LIN {X 0,Y 306.825,Z 754.98,A -85,B 0,C 180,E1 -15915.408,E2 -15915.408} C_VEL
LIN {X 0,Y 305.546,Z 762.411,A -85,B 0,C 180,E1 -15917.38,E2 -15917.38} C_VEL
LIN {X 0,Y 304.708,Z 768.383,A -85,B 0,C 180,E1 -15919.368,E2 -15919.368} C_VEL
LIN {X 0,Y 304.145,Z 773.106,A -85,B 0,C 180,E1 -15921.363,E2 -15921.363} C_VEL
LIN {X 0,Y 303.739,Z 776.717,A -85,B 0,C 180,E1 -15923.358,E2 -15923.358} C_VEL
LIN {X 0,Y 303.637,Z 778.581,A -85,B 0,C 180,E1 -15924.689,E2 -15924.689} C_VEL
LIN {X 0,Y 303.631,Z 779.979,A -85,B 0,C 180,E1 -15926.019,E2 -15926.019} C_VEL
LIN {X 0,Y 303.607,Z 780.975,A -85,B 0,C 180,E1 -15927.348,E2 -15927.348} C_VEL
LIN {X 0,Y 303.564,Z 781.589,A -85,B 0,C 180,E1 -15928.675,E2 -15928.675} C_VEL
LIN {X 0,Y 303.543,Z 783.849,A -85,B 0,C 180,E1 -15931.328,E2 -15931.328} C_VEL
LIN {X 0,Y 303.613,Z 784.204,A -85,B 0,C 180,E1 -15932.655,E2 -15932.655} C_VEL
LIN {X 0,Y 303.689,Z 783.949,A -85,B 0,C 180,E1 -15933.982,E2 -15933.982} C_VEL
LIN {X 0,Y 303.902,Z 782.447,A -85,B 0,C 180,E1 -15936.058,E2 -15936.058} C_VEL
LIN {X 0,Y 304.24,Z 779.671,A -85,B 0,C 180,E1 -15937.968,E2 -15937.968} C_VEL
LIN {X 0,Y 304.907,Z 775.432,A -85,B 0,C 180,E1 -15939.956,E2 -15939.956} C_VEL
LIN {X 0,Y 305.723,Z 769.513,A -85,B 0,C 180,E1 -15941.941,E2 -15941.941} C_VEL
LIN {X 0,Y 306.312,Z 764.494,A -85,B 0,C 180,E1 -15943.265,E2 -15943.265} C_VEL
LIN {X 0,Y 307.414,Z 756.689,A -85,B 0,C 180,E1 -15944.905,E2 -15944.905} C_VEL
LIN {X 0,Y 308.373,Z 747.222,A -85,B 0,C 180,E1 -15946.483,E2 -15946.483} C_VEL
LIN {X 0,Y 308.794,Z 741.989,A -85,B 0,C 180,E1 -15947.211,E2 -15947.211} C_VEL
LIN {X 0,Y 310.204,Z 732.695,A -85,B 0,C 180,E1 -15948.665,E2 -15948.665} C_VEL
LIN {X 0,Y 311.896,Z 721.129,A -85,B 0,C 180,E1 -15950.099,E2 -15950.099} C_VEL
LIN {X 0,Y 313.363,Z 709.743,A -85,B 0,C 180,E1 -15951.202,E2 -15951.202} C_VEL
LIN {X 0,Y 314.572,Z 698.034,A -85,B 0,C 180,E1 -15952.063,E2 -15952.063} C_VEL
LIN {X 0,Y 315.64,Z 685.44,A -85,B 0,C 180,E1 -15952.718,E2 -15952.718} C_VEL
LIN {X 0,Y 316.262,Z 672.598,A -85,B 0,C 180,E1 -15953.146,E2 -15953.146} C_VEL
LIN {X 0,Y 317.533,Z 619.147,A -85,B 0,C 180,E1 -15954.372,E2 -15954.372} C_VEL
LIN {X 0,Y 319.338,Z 611.037,A -85,B 0,C 180,E1 -15955.032,E2 -15955.032} C_VEL
LIN {X 0,Y 321.692,Z 593.032,A -85,B 0,C 180,E1 -15957.134,E2 -15957.134} C_VEL
LIN {X 0,Y 321.832,Z 587.078,A -85,B 0,C 180,E1 -15958.099,E2 -15958.099} C_VEL
LIN {X 0,Y 321.31,Z 583.094,A -85,B 0,C 180,E1 -15958.964,E2 -15958.964} C_VEL
LIN {X 0,Y 320.097,Z 575.053,A -85,B 0,C 180,E1 -15961.099,E2 -15961.099} C_VEL
LIN {X 0,Y 319.576,Z 571.128,A -85,B 0,C 180,E1 -15962.355,E2 -15962.355} C_VEL
LIN {X 0,Y 318.499,Z 569.11,A -85,B 0,C 180,E1 -15963.481,E2 -15963.481} C_VEL
LIN {X 0,Y 317.152,Z 566.664,A -85,B 0,C 180,E1 -15965.181,E2 -15965.181} C_VEL
LIN {X 0,Y 316.078,Z 565.019,A -85,B 0,C 180,E1 -15966.896,E2 -15966.896} C_VEL
LIN {X 0,Y 315.22,Z 564.079,A -85,B 0,C 180,E1 -15968.708,E2 -15968.708} C_VEL
LIN {X 0,Y 314.759,Z 563.673,A -85,B 0,C 180,E1 -15970.61,E2 -15970.61} C_VEL
LIN {X 0,Y 314.997,Z 564.269,A -85,B 0,C 180,E1 -15973.762,E2 -15973.762} C_VEL
LIN {X 0,Y 315.704,Z 566.324,A -85,B 0,C 180,E1 -15976.362,E2 -15976.362} C_VEL
LIN {X 0,Y 316.93,Z 569.514,A -85,B 0,C 180,E1 -15978.936,E2 -15978.936} C_VEL
LIN {X 0,Y 318.658,Z 574.729,A -85,B 0,C 180,E1 -15981.863,E2 -15981.863} C_VEL
LIN {X 0,Y 320.123,Z 580.476,A -85,B 0,C 180,E1 -15984.323,E2 -15984.323} C_VEL
LIN {X 0,Y 321.256,Z 585.775,A -85,B 0,C 180,E1 -15986.235,E2 -15986.235} C_VEL
LIN {X 0,Y 322.064,Z 591.78,A -85,B 0,C 180,E1 -15988.104,E2 -15988.104} C_VEL
LIN {X 0,Y 321.886,Z 594.252,A -85,B 0,C 180,E1 -15988.719,E2 -15988.719} C_VEL
LIN {X 0,Y 317.742,Z 616.41,A -85,B 0,C 180,E1 -15993.422,E2 -15993.422} C_VEL
LIN {X 0,Y 315.354,Z 632.652,A -85,B 0,C 180,E1 -15996.739,E2 -15996.739} C_VEL
LIN {X 0,Y 318.091,Z 647.204,A -85,B 0,C 180,E1 -15997.92,E2 -15997.92} C_VEL
LIN {X 0,Y 319.528,Z 659.288,A -85,B 0,C 180,E1 -15998.728,E2 -15998.728} C_VEL
LIN {X 0,Y 316.266,Z 706.91,A -85,B 0,C 180,E1 -16000.529,E2 -16000.529} C_VEL
LIN {X 0,Y 315.093,Z 718.743,A -85,B 0,C 180,E1 -16001.215,E2 -16001.215} C_VEL
LIN {X 0,Y 313.817,Z 728.863,A -85,B 0,C 180,E1 -16002.065,E2 -16002.065} C_VEL
LIN {X 0,Y 312.287,Z 738.973,A -85,B 0,C 180,E1 -16003.157,E2 -16003.157} C_VEL
LIN {X 0,Y 310.981,Z 746.942,A -85,B 0,C 180,E1 -16004.265,E2 -16004.265} C_VEL
LIN {X 0,Y 309.584,Z 754.286,A -85,B 0,C 180,E1 -16005.539,E2 -16005.539} C_VEL
LIN {X 0,Y 308.32,Z 760.339,A -85,B 0,C 180,E1 -16006.824,E2 -16006.824} C_VEL
LIN {X 0,Y 307.008,Z 766.483,A -85,B 0,C 180,E1 -16008.445,E2 -16008.445} C_VEL
LIN {X 0,Y 305.966,Z 771.229,A -85,B 0,C 180,E1 -16010.08,E2 -16010.08} C_VEL
LIN {X 0,Y 305.24,Z 774.224,A -85,B 0,C 180,E1 -16011.393,E2 -16011.393} C_VEL
LIN {X 0,Y 304.609,Z 777.366,A -85,B 0,C 180,E1 -16013.376,E2 -16013.376} C_VEL
LIN {X 0,Y 304.172,Z 778.748,A -85,B 0,C 180,E1 -16014.697,E2 -16014.697} C_VEL
LIN {X 0,Y 303.852,Z 779.547,A -85,B 0,C 180,E1 -16016.021,E2 -16016.021} C_VEL
LIN {X 0,Y 303.664,Z 779.771,A -85,B 0,C 180,E1 -16017.347,E2 -16017.347} C_VEL
LIN {X 0,Y 303.55,Z 779.388,A -85,B 0,C 180,E1 -16018.673,E2 -16018.673} C_VEL
LIN {X 0,Y 303.534,Z 778.387,A -85,B 0,C 180,E1 -16020,E2 -16020} C_VEL
LIN {X 0,Y 303.571,Z 775.717,A -85,B 0,C 180,E1 -16021.99,E2 -16021.99} C_VEL
LIN {X 0,Y 303.815,Z 771.583,A -85,B 0,C 180,E1 -16023.979,E2 -16023.979} C_VEL
LIN {X 0,Y 303.878,Z 765.594,A -85,B 0,C 180,E1 -16026.01,E2 -16026.01} C_VEL
LIN {X 0,Y 304.246,Z 759.517,A -85,B 0,C 180,E1 -16027.571,E2 -16027.571} C_VEL
LIN {X 0,Y 304.58,Z 752.814,A -85,B 0,C 180,E1 -16028.961,E2 -16028.961} C_VEL
LIN {X 0,Y 305.028,Z 744.827,A -85,B 0,C 180,E1 -16030.286,E2 -16030.286} C_VEL
LIN {X 0,Y 305.485,Z 736.01,A -85,B 0,C 180,E1 -16031.445,E2 -16031.445} C_VEL
LIN {X 0,Y 305.984,Z 726.568,A -85,B 0,C 180,E1 -16032.435,E2 -16032.435} C_VEL
LIN {X 0,Y 306.384,Z 715.842,A -85,B 0,C 180,E1 -16033.261,E2 -16033.261} C_VEL
LIN {X 0,Y 306.839,Z 705.379,A -85,B 0,C 180,E1 -16033.832,E2 -16033.832} C_VEL
LIN {X 0,Y 307.924,Z 653.383,A -85,B 0,C 180,E1 -16035.606,E2 -16035.606} C_VEL
LIN {X 0,Y 306.354,Z 631.88,A -85,B 0,C 180,E1 -16036.403,E2 -16036.403} C_VEL
LIN {X 0,Y 307.681,Z 611.142,A -85,B 0,C 180,E1 -16040.383,E2 -16040.383} C_VEL
LIN {X 0,Y 309.256,Z 588.247,A -85,B 0,C 180,E1 -16044.799,E2 -16044.799} C_VEL
LIN {X 0,Y 310.552,Z 571.445,A -85,B 0,C 180,E1 -16048.041,E2 -16048.041} C_VEL
LIN {X 0,Y 308.725,Z 561.43,A -85,B 0,C 180,E1 -16050.11,E2 -16050.11} C_VEL
LIN {X 0,Y 305.543,Z 546.572,A -85,B 0,C 180,E1 -16053.314,E2 -16053.314} C_VEL
LIN {X 0,Y 305.48,Z 546.435,A -85,B 0,C 180,E1 -16056.739,E2 -16056.739} C_VEL
LIN {X 0,Y 305.459,Z 546.414,A -85,B 0,C 180,E1 -16060.599,E2 -16060.599} C_VEL
LIN {X 0,Y 305.431,Z 546.409,A -85,B 0,C 180,E1 -16064.494,E2 -16064.494} C_VEL
LIN {X 0,Y 305.48,Z 546.425,A -85,B 0,C 180,E1 -16068.149,E2 -16068.149} C_VEL
LIN {X 0,Y 305.472,Z 546.41,A -85,B 0,C 180,E1 -16071.596,E2 -16071.596} C_VEL
LIN {X 0,Y 305.467,Z 546.424,A -85,B 0,C 180,E1 -16074.886,E2 -16074.886} C_VEL
LIN {X 0,Y 305.456,Z 546.43,A -85,B 0,C 180,E1 -16078.354,E2 -16078.354} C_VEL
LIN {X 0,Y 305.535,Z 546.476,A -85,B 0,C 180,E1 -16080.803,E2 -16080.803} C_VEL
LIN {X 0,Y 307.121,Z 553.574,A -85,B 0,C 180,E1 -16083.444,E2 -16083.444} C_VEL
LIN {X 0,Y 307.557,Z 555.026,A -85,B 0,C 180,E1 -16083.632,E2 -16083.632} C_VEL
LIN {X 0,Y 314.364,Z 571.514,A -85,B 0,C 180,E1 -16084.671,E2 -16084.671} C_VEL
LIN {X 0,Y 316.455,Z 577.195,A -85,B 0,C 180,E1 -16084.992,E2 -16084.992} C_VEL
LIN {X 0,Y 318.23,Z 587.121,A -85,B 0,C 180,E1 -16085.384,E2 -16085.384} C_VEL
LIN {X 0,Y 316.373,Z 660.195,A -85,B 0,C 180,E1 -16087.036,E2 -16087.036} C_VEL
LIN {X 0,Y 315.644,Z 673.592,A -85,B 0,C 180,E1 -16087.585,E2 -16087.585} C_VEL
LIN {X 0,Y 314.69,Z 686.351,A -85,B 0,C 180,E1 -16088.376,E2 -16088.376} C_VEL
LIN {X 0,Y 313.452,Z 697.672,A -85,B 0,C 180,E1 -16089.32,E2 -16089.32} C_VEL
LIN {X 0,Y 311.954,Z 709.318,A -85,B 0,C 180,E1 -16090.59,E2 -16090.59} C_VEL
LIN {X 0,Y 310.534,Z 720.204,A -85,B 0,C 180,E1 -16092.108,E2 -16092.108} C_VEL
LIN {X 0,Y 309.013,Z 729.997,A -85,B 0,C 180,E1 -16093.822,E2 -16093.822} C_VEL
LIN {X 0,Y 307.427,Z 738.909,A -85,B 0,C 180,E1 -16095.773,E2 -16095.773} C_VEL
LIN {X 0,Y 306.273,Z 746.076,A -85,B 0,C 180,E1 -16097.744,E2 -16097.744} C_VEL
LIN {X 0,Y 305.411,Z 750.913,A -85,B 0,C 180,E1 -16099.391,E2 -16099.391} C_VEL
LIN {X 0,Y 304.679,Z 755.609,A -85,B 0,C 180,E1 -16101.376,E2 -16101.376} C_VEL
LIN {X 0,Y 304.196,Z 759.318,A -85,B 0,C 180,E1 -16103.442,E2 -16103.442} C_VEL
LIN {X 0,Y 304.024,Z 761.05,A -85,B 0,C 180,E1 -16104.693,E2 -16104.693} C_VEL
LIN {X 0,Y 303.867,Z 762.446,A -85,B 0,C 180,E1 -16106.02,E2 -16106.02} C_VEL
LIN {X 0,Y 303.617,Z 764.054,A -85,B 0,C 180,E1 -16108.672,E2 -16108.672} C_VEL
LIN {X 0,Y 303.611,Z 764.285,A -85,B 0,C 180,E1 -16109.999,E2 -16109.999} C_VEL
LIN {X 0,Y 303.617,Z 764.095,A -85,B 0,C 180,E1 -16111.325,E2 -16111.325} C_VEL
LIN {X 0,Y 303.862,Z 762.543,A -85,B 0,C 180,E1 -16113.978,E2 -16113.978} C_VEL
LIN {X 0,Y 304.019,Z 761.188,A -85,B 0,C 180,E1 -16115.304,E2 -16115.304} C_VEL
LIN {X 0,Y 304.345,Z 758.321,A -85,B 0,C 180,E1 -16117.295,E2 -16117.295} C_VEL
LIN {X 0,Y 304.844,Z 754.433,A -85,B 0,C 180,E1 -16119.286,E2 -16119.286} C_VEL
LIN {X 0,Y 305.715,Z 749.416,A -85,B 0,C 180,E1 -16121.267,E2 -16121.267} C_VEL
LIN {X 0,Y 306.746,Z 743.101,A -85,B 0,C 180,E1 -16123.244,E2 -16123.244} C_VEL
LIN {X 0,Y 308.104,Z 735.191,A -85,B 0,C 180,E1 -16125.206,E2 -16125.206} C_VEL
LIN {X 0,Y 309.826,Z 725.349,A -85,B 0,C 180,E1 -16127.149,E2 -16127.149} C_VEL
LIN {X 0,Y 311.239,Z 715.021,A -85,B 0,C 180,E1 -16128.769,E2 -16128.769} C_VEL
LIN {X 0,Y 312.599,Z 704.79,A -85,B 0,C 180,E1 -16130.05,E2 -16130.05} C_VEL
LIN {X 0,Y 313.983,Z 693.583,A -85,B 0,C 180,E1 -16131.156,E2 -16131.156} C_VEL
LIN {X 0,Y 315.21,Z 680.94,A -85,B 0,C 180,E1 -16132.1,E2 -16132.1} C_VEL
LIN {X 0,Y 316.045,Z 668.274,A -85,B 0,C 180,E1 -16132.771,E2 -16132.771} C_VEL
LIN {X 0,Y 316.658,Z 655.229,A -85,B 0,C 180,E1 -16133.199,E2 -16133.199} C_VEL
LIN {X 0,Y 318.19,Z 585.949,A -85,B 0,C 180,E1 -16134.76,E2 -16134.76} C_VEL
LIN {X 0,Y 315.996,Z 575.742,A -85,B 0,C 180,E1 -16135.197,E2 -16135.197} C_VEL
LIN {X 0,Y 309.077,Z 558.611,A -85,B 0,C 180,E1 -16136.241,E2 -16136.241} C_VEL
LIN {X 0,Y 307.194,Z 553.882,A -85,B 0,C 180,E1 -16136.597,E2 -16136.597} C_VEL
LIN {X 0,Y 305.932,Z 548.426,A -85,B 0,C 180,E1 -16138.518,E2 -16138.518} C_VEL
LIN {X 0,Y 305.264,Z 547.176,A -85,B 0,C 180,E1 -16139.189,E2 -16139.189} C_VEL
LIN {X 0,Y 304.227,Z 546.692,A -85,B 0,C 180,E1 -16139.887,E2 -16139.887} C_VEL
LIN {X 0,Y 299.362,Z 547.224,A -85,B 0,C 180,E1 -16142.794,E2 -16142.794} C_VEL
LIN {X 0,Y 298.448,Z 547.31,A -85,B 0,C 180,E1 -16143.945,E2 -16143.945} C_VEL
LIN {X 0,Y 298.4,Z 547.316,A -85,B 0,C 180,E1 -16144.333,E2 -16144.333} C_VEL
LIN {X 0,Y 298.433,Z 547.313,A -85,B 0,C 180,E1 -16147.753,E2 -16147.753} C_VEL
LIN {X 0,Y 298.382,Z 547.313,A -85,B 0,C 180,E1 -16151.26,E2 -16151.26} C_VEL
LIN {X 0,Y 298.35,Z 547.302,A -85,B 0,C 180,E1 -16155.034,E2 -16155.034} C_VEL
LIN {X 0,Y 298.427,Z 547.307,A -85,B 0,C 180,E1 -16156.925,E2 -16156.925} C_VEL
LIN {X 0,Y 298.421,Z 547.286,A -85,B 0,C 180,E1 -16161,E2 -16161} C_VEL
LIN {X 0,Y 298.43,Z 547.307,A -85,B 0,C 180,E1 -16163.932,E2 -16163.932} C_VEL
LIN {X 0,Y 298.39,Z 547.31,A -85,B 0,C 180,E1 -16167.982,E2 -16167.982} C_VEL
LIN {X 0,Y 298.457,Z 547.297,A -85,B 0,C 180,E1 -16171.904,E2 -16171.904} C_VEL
LIN {X 0,Y 298.479,Z 547.304,A -85,B 0,C 180,E1 -16174.923,E2 -16174.923} C_VEL
LIN {X 0,Y 298.443,Z 547.303,A -85,B 0,C 180,E1 -16179.315,E2 -16179.315} C_VEL
LIN {X 0,Y 298.531,Z 547.292,A -85,B 0,C 180,E1 -16182.179,E2 -16182.179} C_VEL
LIN {X 0,Y 298.586,Z 547.281,A -85,B 0,C 180,E1 -16184.994,E2 -16184.994} C_VEL
LIN {X 0,Y 298.586,Z 547.281,A -85,B 0,C 180,E1 -16189.146,E2 -16189.146} C_VEL
LIN {X 0,Y 298.751,Z 547.266,A -85,B 0,C 180,E1 -16191.886,E2 -16191.886} C_VEL
LIN {X 0,Y 298.654,Z 547.28,A -85,B 0,C 180,E1 -16194.599,E2 -16194.599} C_VEL
LIN {X 0,Y 298.918,Z 547.244,A -85,B 0,C 180,E1 -16198.653,E2 -16198.653} C_VEL
LIN {X 0,Y 298.918,Z 547.249,A -85,B 0,C 180,E1 -16201.347,E2 -16201.347} C_VEL
LIN {X 0,Y 298.792,Z 547.264,A -85,B 0,C 180,E1 -16206.754,E2 -16206.754} C_VEL
LIN {X 0,Y 298.673,Z 547.268,A -85,B 0,C 180,E1 -16209.481,E2 -16209.481} C_VEL
LIN {X 0,Y 298.546,Z 547.297,A -85,B 0,C 180,E1 -16213.616,E2 -16213.616} C_VEL
LIN {X 0,Y 298.541,Z 547.285,A -85,B 0,C 180,E1 -16216.409,E2 -16216.409} C_VEL
LIN {X 0,Y 298.509,Z 547.301,A -85,B 0,C 180,E1 -16219.658,E2 -16219.658} C_VEL
LIN {X 0,Y 298.451,Z 547.308,A -85,B 0,C 180,E1 -16223.598,E2 -16223.598} C_VEL
LIN {X 0,Y 298.477,Z 547.295,A -85,B 0,C 180,E1 -16226.576,E2 -16226.576} C_VEL
LIN {X 0,Y 298.41,Z 547.313,A -85,B 0,C 180,E1 -16229.642,E2 -16229.642} C_VEL
LIN {X 0,Y 298.389,Z 547.315,A -85,B 0,C 180,E1 -16232.801,E2 -16232.801} C_VEL
LIN {X 0,Y 298.441,Z 547.284,A -85,B 0,C 180,E1 -16236.809,E2 -16236.809} C_VEL
LIN {X 0,Y 298.409,Z 547.305,A -85,B 0,C 180,E1 -16241.258,E2 -16241.258} C_VEL
LIN {X 0,Y 298.412,Z 547.314,A -85,B 0,C 180,E1 -16245.048,E2 -16245.048} C_VEL
LIN {X 0,Y 298.45,Z 547.309,A -85,B 0,C 180,E1 -16248.751,E2 -16248.751} C_VEL
LIN {X 0,Y 298.463,Z 547.279,A -85,B 0,C 180,E1 -16253.189,E2 -16253.189} C_VEL
LIN {X 0,Y 298.426,Z 547.398,A -85,B 0,C 180,E1 -16255.789,E2 -16255.789} C_VEL
LIN {X 0,Y 300.553,Z 556.606,A -85,B 0,C 180,E1 -16259.042,E2 -16259.042} C_VEL
LIN {X 0,Y 302.687,Z 566.604,A -85,B 0,C 180,E1 -16262.332,E2 -16262.332} C_VEL
LIN {X 0,Y 303.149,Z 569.151,A -85,B 0,C 180,E1 -16263.067,E2 -16263.067} C_VEL
LIN {X 0,Y 305.199,Z 575.225,A -85,B 0,C 180,E1 -16263.464,E2 -16263.464} C_VEL
LIN {X 0,Y 310.189,Z 604.18,A -85,B 0,C 180,E1 -16264.648,E2 -16264.648} C_VEL
LIN {X 0,Y 311.262,Z 612.409,A -85,B 0,C 180,E1 -16264.946,E2 -16264.946} C_VEL
LIN {X 0,Y 309.607,Z 677.501,A -85,B 0,C 180,E1 -16266.462,E2 -16266.462} C_VEL
LIN {X 0,Y 308.607,Z 691.422,A -85,B 0,C 180,E1 -16267.047,E2 -16267.047} C_VEL
LIN {X 0,Y 307.431,Z 703.883,A -85,B 0,C 180,E1 -16267.841,E2 -16267.841} C_VEL
LIN {X 0,Y 306.08,Z 715.003,A -85,B 0,C 180,E1 -16268.8,E2 -16268.8} C_VEL
LIN {X 0,Y 304.44,Z 726.577,A -85,B 0,C 180,E1 -16270.094,E2 -16270.094} C_VEL
LIN {X 0,Y 302.776,Z 737,A -85,B 0,C 180,E1 -16271.564,E2 -16271.564} C_VEL
LIN {X 0,Y 301.509,Z 745.549,A -85,B 0,C 180,E1 -16273.065,E2 -16273.065} C_VEL
LIN {X 0,Y 300.188,Z 753.4,A -85,B 0,C 180,E1 -16274.73,E2 -16274.73} C_VEL
LIN {X 0,Y 298.808,Z 761.087,A -85,B 0,C 180,E1 -16276.744,E2 -16276.744} C_VEL
LIN {X 0,Y 297.712,Z 768.179,A -85,B 0,C 180,E1 -16279.115,E2 -16279.115} C_VEL
LIN {X 0,Y 297.087,Z 772.901,A -85,B 0,C 180,E1 -16281.156,E2 -16281.156} C_VEL
LIN {X 0,Y 296.686,Z 776.513,A -85,B 0,C 180,E1 -16283.199,E2 -16283.199} C_VEL
LIN {X 0,Y 296.552,Z 778.377,A -85,B 0,C 180,E1 -16284.562,E2 -16284.562} C_VEL
LIN {X 0,Y 296.528,Z 779.774,A -85,B 0,C 180,E1 -16285.924,E2 -16285.924} C_VEL
LIN {X 0,Y 296.533,Z 780.771,A -85,B 0,C 180,E1 -16287.284,E2 -16287.284} C_VEL
LIN {X 0,Y 296.484,Z 781.379,A -85,B 0,C 180,E1 -16288.643,E2 -16288.643} C_VEL
LIN {X 0,Y 296.465,Z 783.587,A -85,B 0,C 180,E1 -16291.36,E2 -16291.36} C_VEL
LIN {X 0,Y 296.541,Z 784.068,A -85,B 0,C 180,E1 -16292.718,E2 -16292.718} C_VEL
LIN {X 0,Y 296.591,Z 783.961,A -85,B 0,C 180,E1 -16294.078,E2 -16294.078} C_VEL
LIN {X 0,Y 296.821,Z 782.819,A -85,B 0,C 180,E1 -16296.033,E2 -16296.033} C_VEL
LIN {X 0,Y 297.23,Z 780.165,A -85,B 0,C 180,E1 -16298.157,E2 -16298.157} C_VEL
LIN {X 0,Y 297.681,Z 777.674,A -85,B 0,C 180,E1 -16299.514,E2 -16299.514} C_VEL
LIN {X 0,Y 298.212,Z 774.484,A -85,B 0,C 180,E1 -16300.869,E2 -16300.869} C_VEL
LIN {X 0,Y 299.015,Z 769.366,A -85,B 0,C 180,E1 -16302.558,E2 -16302.558} C_VEL
LIN {X 0,Y 299.803,Z 764.371,A -85,B 0,C 180,E1 -16303.904,E2 -16303.904} C_VEL
LIN {X 0,Y 300.94,Z 756.662,A -85,B 0,C 180,E1 -16305.58,E2 -16305.58} C_VEL
LIN {X 0,Y 302.009,Z 747.777,A -85,B 0,C 180,E1 -16307.097,E2 -16307.097} C_VEL
LIN {X 0,Y 302.796,Z 738.445,A -85,B 0,C 180,E1 -16308.384,E2 -16308.384} C_VEL
LIN {X 0,Y 303.445,Z 732.497,A -85,B 0,C 180,E1 -16309.097,E2 -16309.097} C_VEL
LIN {X 0,Y 305.028,Z 722.348,A -85,B 0,C 180,E1 -16310.396,E2 -16310.396} C_VEL
LIN {X 0,Y 306.516,Z 711.301,A -85,B 0,C 180,E1 -16311.523,E2 -16311.523} C_VEL
LIN {X 0,Y 307.889,Z 699.055,A -85,B 0,C 180,E1 -16312.48,E2 -16312.48} C_VEL
LIN {X 0,Y 308.997,Z 687.058,A -85,B 0,C 180,E1 -16313.146,E2 -16313.146} C_VEL
LIN {X 0,Y 309.703,Z 673.882,A -85,B 0,C 180,E1 -16313.621,E2 -16313.621} C_VEL
LIN {X 0,Y 310.962,Z 625.82,A -85,B 0,C 180,E1 -16314.761,E2 -16314.761} C_VEL
LIN {X 0,Y 314.172,Z 612.643,A -85,B 0,C 180,E1 -16315.862,E2 -16315.862} C_VEL
LIN {X 0,Y 316.645,Z 596.601,A -85,B 0,C 180,E1 -16317.782,E2 -16317.782} C_VEL
LIN {X 0,Y 316.946,Z 590.536,A -85,B 0,C 180,E1 -16318.788,E2 -16318.788} C_VEL
LIN {X 0,Y 316.071,Z 583.822,A -85,B 0,C 180,E1 -16320.453,E2 -16320.453} C_VEL
LIN {X 0,Y 315.334,Z 577.432,A -85,B 0,C 180,E1 -16322.338,E2 -16322.338} C_VEL
LIN {X 0,Y 315.02,Z 576.052,A -85,B 0,C 180,E1 -16322.881,E2 -16322.881} C_VEL
LIN {X 0,Y 313.397,Z 573.124,A -85,B 0,C 180,E1 -16324.757,E2 -16324.757} C_VEL
LIN {X 0,Y 312.55,Z 571.715,A -85,B 0,C 180,E1 -16325.953,E2 -16325.953} C_VEL
LIN {X 0,Y 311.446,Z 570.264,A -85,B 0,C 180,E1 -16327.833,E2 -16327.833} C_VEL
LIN {X 0,Y 310.711,Z 569.522,A -85,B 0,C 180,E1 -16329.731,E2 -16329.731} C_VEL
LIN {X 0,Y 310.497,Z 569.555,A -85,B 0,C 180,E1 -16332.77,E2 -16332.77} C_VEL
LIN {X 0,Y 310.771,Z 570.278,A -85,B 0,C 180,E1 -16334.513,E2 -16334.513} C_VEL
LIN {X 0,Y 311.578,Z 572.968,A -85,B 0,C 180,E1 -16337.415,E2 -16337.415} C_VEL
LIN {X 0,Y 312.662,Z 576.349,A -85,B 0,C 180,E1 -16339.842,E2 -16339.842} C_VEL
LIN {X 0,Y 313.856,Z 580.516,A -85,B 0,C 180,E1 -16342.117,E2 -16342.117} C_VEL
LIN {X 0,Y 315.36,Z 587.458,A -85,B 0,C 180,E1 -16345.029,E2 -16345.029} C_VEL
LIN {X 0,Y 316.237,Z 593.305,A -85,B 0,C 180,E1 -16347.045,E2 -16347.045} C_VEL
LIN {X 0,Y 316.318,Z 596.748,A -85,B 0,C 180,E1 -16348.053,E2 -16348.053} C_VEL
LIN {X 0,Y 312.172,Z 617.259,A -85,B 0,C 180,E1 -16352.515,E2 -16352.515} C_VEL
LIN {X 0,Y 309.562,Z 632.55,A -85,B 0,C 180,E1 -16355.74,E2 -16355.74} C_VEL
LIN {X 0,Y 312.365,Z 647.726,A -85,B 0,C 180,E1 -16357.07,E2 -16357.07} C_VEL
LIN {X 0,Y 313.908,Z 660.09,A -85,B 0,C 180,E1 -16357.941,E2 -16357.941} C_VEL
LIN {X 0,Y 310.383,Z 707.099,A -85,B 0,C 180,E1 -16359.8,E2 -16359.8} C_VEL
LIN {X 0,Y 309.16,Z 718.874,A -85,B 0,C 180,E1 -16360.495,E2 -16360.495} C_VEL
LIN {X 0,Y 307.79,Z 728.991,A -85,B 0,C 180,E1 -16361.357,E2 -16361.357} C_VEL
LIN {X 0,Y 306.381,Z 737.697,A -85,B 0,C 180,E1 -16362.306,E2 -16362.306} C_VEL
LIN {X 0,Y 304.711,Z 746.945,A -85,B 0,C 180,E1 -16363.588,E2 -16363.588} C_VEL
LIN {X 0,Y 303.217,Z 754.234,A -85,B 0,C 180,E1 -16364.885,E2 -16364.885} C_VEL
LIN {X 0,Y 301.835,Z 760.322,A -85,B 0,C 180,E1 -16366.192,E2 -16366.192} C_VEL
LIN {X 0,Y 300.363,Z 766.508,A -85,B 0,C 180,E1 -16367.843,E2 -16367.843} C_VEL
LIN {X 0,Y 299.433,Z 770.408,A -85,B 0,C 180,E1 -16369.177,E2 -16369.177} C_VEL
LIN {X 0,Y 298.252,Z 774.825,A -85,B 0,C 180,E1 -16371.19,E2 -16371.19} C_VEL
LIN {X 0,Y 297.841,Z 776.718,A -85,B 0,C 180,E1 -16372.335,E2 -16372.335} C_VEL
LIN {X 0,Y 297.119,Z 779.033,A -85,B 0,C 180,E1 -16374.571,E2 -16374.571} C_VEL
LIN {X 0,Y 296.779,Z 779.685,A -85,B 0,C 180,E1 -16375.926,E2 -16375.926} C_VEL
LIN {X 0,Y 296.596,Z 779.76,A -85,B 0,C 180,E1 -16377.284,E2 -16377.284} C_VEL
LIN {X 0,Y 296.473,Z 779.257,A -85,B 0,C 180,E1 -16378.642,E2 -16378.642} C_VEL
LIN {X 0,Y 296.453,Z 778.164,A -85,B 0,C 180,E1 -16380,E2 -16380} C_VEL
LIN {X 0,Y 296.498,Z 775.28,A -85,B 0,C 180,E1 -16382.038,E2 -16382.038} C_VEL
LIN {X 0,Y 296.662,Z 772.566,A -85,B 0,C 180,E1 -16383.395,E2 -16383.395} C_VEL
LIN {X 0,Y 296.724,Z 769.093,A -85,B 0,C 180,E1 -16384.755,E2 -16384.755} C_VEL
LIN {X 0,Y 296.906,Z 763.827,A -85,B 0,C 180,E1 -16386.387,E2 -16386.387} C_VEL
LIN {X 0,Y 297.302,Z 756.526,A -85,B 0,C 180,E1 -16388.154,E2 -16388.154} C_VEL
LIN {X 0,Y 297.735,Z 748.342,A -85,B 0,C 180,E1 -16389.682,E2 -16389.682} C_VEL
LIN {X 0,Y 298.236,Z 739.254,A -85,B 0,C 180,E1 -16391.039,E2 -16391.039} C_VEL
LIN {X 0,Y 298.728,Z 730.472,A -85,B 0,C 180,E1 -16392.052,E2 -16392.052} C_VEL
LIN {X 0,Y 299.193,Z 720.194,A -85,B 0,C 180,E1 -16392.981,E2 -16392.981} C_VEL
LIN {X 0,Y 299.598,Z 708.276,A -85,B 0,C 180,E1 -16393.74,E2 -16393.74} C_VEL
LIN {X 0,Y 299.891,Z 696,A -85,B 0,C 180,E1 -16394.245,E2 -16394.245} C_VEL
LIN {X 0,Y 300.836,Z 653.46,A -85,B 0,C 180,E1 -16395.735,E2 -16395.735} C_VEL
LIN {X 0,Y 299.295,Z 632.005,A -85,B 0,C 180,E1 -16396.542,E2 -16396.542} C_VEL
LIN {X 0,Y 300.51,Z 613.304,A -85,B 0,C 180,E1 -16400.179,E2 -16400.179} C_VEL
LIN {X 0,Y 301.91,Z 593.601,A -85,B 0,C 180,E1 -16404.04,E2 -16404.04} C_VEL
LIN {X 0,Y 303.572,Z 572.993,A -85,B 0,C 180,E1 -16408.08,E2 -16408.08} C_VEL
LIN {X 0,Y 302.429,Z 565.89,A -85,B 0,C 180,E1 -16409.556,E2 -16409.556} C_VEL
LIN {X 0,Y 298.859,Z 549.228,A -85,B 0,C 180,E1 -16413.145,E2 -16413.145} C_VEL
LIN {X 0,Y 298.463,Z 547.434,A -85,B 0,C 180,E1 -16413.598,E2 -16413.598} C_VEL
LIN {X 0,Y 298.429,Z 547.311,A -85,B 0,C 180,E1 -16417.756,E2 -16417.756} C_VEL
LIN {X 0,Y 298.389,Z 547.282,A -85,B 0,C 180,E1 -16421.261,E2 -16421.261} C_VEL
LIN {X 0,Y 298.393,Z 547.294,A -85,B 0,C 180,E1 -16425.041,E2 -16425.041} C_VEL
LIN {X 0,Y 298.422,Z 547.296,A -85,B 0,C 180,E1 -16428.743,E2 -16428.743} C_VEL
LIN {X 0,Y 298.449,Z 547.31,A -85,B 0,C 180,E1 -16433.192,E2 -16433.192} C_VEL
LIN {X 0,Y 298.4,Z 547.317,A -85,B 0,C 180,E1 -16437.199,E2 -16437.199} C_VEL
LIN {X 0,Y 298.487,Z 547.465,A -85,B 0,C 180,E1 -16440.365,E2 -16440.365} C_VEL
LIN {X 0,Y 300.019,Z 554.106,A -85,B 0,C 180,E1 -16442.831,E2 -16442.831} C_VEL
LIN {X 0,Y 302.339,Z 559.625,A -85,B 0,C 180,E1 -16443.267,E2 -16443.267} C_VEL
LIN {X 0,Y 309.127,Z 576.367,A -85,B 0,C 180,E1 -16444.329,E2 -16444.329} C_VEL
LIN {X 0,Y 310.52,Z 580.766,A -85,B 0,C 180,E1 -16444.564,E2 -16444.564} C_VEL
LIN {X 0,Y 311.778,Z 588.203,A -85,B 0,C 180,E1 -16444.861,E2 -16444.861} C_VEL
LIN {X 0,Y 309.867,Z 660.416,A -85,B 0,C 180,E1 -16446.525,E2 -16446.525} C_VEL
LIN {X 0,Y 309.085,Z 673.808,A -85,B 0,C 180,E1 -16447.082,E2 -16447.082} C_VEL
LIN {X 0,Y 308.101,Z 686.563,A -85,B 0,C 180,E1 -16447.89,E2 -16447.89} C_VEL
LIN {X 0,Y 306.822,Z 697.882,A -85,B 0,C 180,E1 -16448.852,E2 -16448.852} C_VEL
LIN {X 0,Y 305.261,Z 709.527,A -85,B 0,C 180,E1 -16450.147,E2 -16450.147} C_VEL
LIN {X 0,Y 303.745,Z 720.414,A -85,B 0,C 180,E1 -16451.694,E2 -16451.694} C_VEL
LIN {X 0,Y 302.185,Z 730.205,A -85,B 0,C 180,E1 -16453.446,E2 -16453.446} C_VEL
LIN {X 0,Y 300.558,Z 739.116,A -85,B 0,C 180,E1 -16455.44,E2 -16455.44} C_VEL
LIN {X 0,Y 299.318,Z 746.283,A -85,B 0,C 180,E1 -16457.455,E2 -16457.455} C_VEL
LIN {X 0,Y 298.438,Z 751.119,A -85,B 0,C 180,E1 -16459.14,E2 -16459.14} C_VEL
LIN {X 0,Y 297.638,Z 755.815,A -85,B 0,C 180,E1 -16461.17,E2 -16461.17} C_VEL
LIN {X 0,Y 297.119,Z 759.774,A -85,B 0,C 180,E1 -16463.447,E2 -16463.447} C_VEL
LIN {X 0,Y 296.785,Z 762.651,A -85,B 0,C 180,E1 -16465.925,E2 -16465.925} C_VEL
LIN {X 0,Y 296.536,Z 764.258,A -85,B 0,C 180,E1 -16468.641,E2 -16468.641} C_VEL
LIN {X 0,Y 296.526,Z 764.49,A -85,B 0,C 180,E1 -16469.999,E2 -16469.999} C_VEL
LIN {X 0,Y 296.535,Z 764.299,A -85,B 0,C 180,E1 -16471.357,E2 -16471.357} C_VEL
LIN {X 0,Y 296.78,Z 762.747,A -85,B 0,C 180,E1 -16474.073,E2 -16474.073} C_VEL
LIN {X 0,Y 297.09,Z 760.011,A -85,B 0,C 180,E1 -16476.504,E2 -16476.504} C_VEL
LIN {X 0,Y 297.635,Z 756.05,A -85,B 0,C 180,E1 -16478.828,E2 -16478.828} C_VEL
LIN {X 0,Y 298.411,Z 751.418,A -85,B 0,C 180,E1 -16480.859,E2 -16480.859} C_VEL
LIN {X 0,Y 299.656,Z 744.434,A -85,B 0,C 180,E1 -16483.218,E2 -16483.218} C_VEL
LIN {X 0,Y 300.977,Z 736.862,A -85,B 0,C 180,E1 -16485.229,E2 -16485.229} C_VEL
LIN {X 0,Y 302.769,Z 727.325,A -85,B 0,C 180,E1 -16487.214,E2 -16487.214} C_VEL
LIN {X 0,Y 304.203,Z 717.486,A -85,B 0,C 180,E1 -16488.87,E2 -16488.87} C_VEL
LIN {X 0,Y 305.559,Z 707.802,A -85,B 0,C 180,E1 -16490.181,E2 -16490.181} C_VEL
LIN {X 0,Y 306.969,Z 697.307,A -85,B 0,C 180,E1 -16491.311,E2 -16491.311} C_VEL
LIN {X 0,Y 308.323,Z 684.656,A -85,B 0,C 180,E1 -16492.356,E2 -16492.356} C_VEL
LIN {X 0,Y 309.287,Z 671.993,A -85,B 0,C 180,E1 -16493.12,E2 -16493.12} C_VEL
LIN {X 0,Y 310.004,Z 659.915,A -85,B 0,C 180,E1 -16493.594,E2 -16493.594} C_VEL
LIN {X 0,Y 311.739,Z 586.94,A -85,B 0,C 180,E1 -16495.288,E2 -16495.288} C_VEL
LIN {X 0,Y 309.882,Z 578.322,A -85,B 0,C 180,E1 -16495.669,E2 -16495.669} C_VEL
LIN {X 0,Y 302.632,Z 560.281,A -85,B 0,C 180,E1 -16496.805,E2 -16496.805} C_VEL
LIN {X 0,Y 300.076,Z 554.221,A -85,B 0,C 180,E1 -16497.262,E2 -16497.262} C_VEL
LIN {X 0,Y 298.491,Z 547.517,A -85,B 0,C 180,E1 -16499.729,E2 -16499.729} C_VEL
LIN {X 0,Y 298.392,Z 547.315,A -85,B 0,C 180,E1 -16502.015,E2 -16502.015} C_VEL
LIN {X 0,Y 298.4,Z 547.316,A -85,B 0,C 180,E1 -16504.333,E2 -16504.333} C_VEL
LIN {X 0,Y 297.795,Z 547.4,A -85,B 0,C 180,E1 -16505.459,E2 -16505.459} C_VEL
LIN {X 0,Y 294.952,Z 547.747,A -85,B 0,C 180,E1 -16507.291,E2 -16507.291} C_VEL
LIN {X 0,Y 292.494,Z 548.045,A -85,B 0,C 180,E1 -16508.779,E2 -16508.779} C_VEL
LIN {X 0,Y 291.426,Z 548.171,A -85,B 0,C 180,E1 -16509.931,E2 -16509.931} C_VEL
LIN {X 0,Y 291.335,Z 548.183,A -85,B 0,C 180,E1 -16510.322,E2 -16510.322} C_VEL
LIN {X 0,Y 291.285,Z 548.183,A -85,B 0,C 180,E1 -16514.401,E2 -16514.401} C_VEL
LIN {X 0,Y 291.351,Z 548.192,A -85,B 0,C 180,E1 -16518.397,E2 -16518.397} C_VEL
LIN {X 0,Y 291.37,Z 548.163,A -85,B 0,C 180,E1 -16521.161,E2 -16521.161} C_VEL
LIN {X 0,Y 291.381,Z 548.188,A -85,B 0,C 180,E1 -16524.629,E2 -16524.629} C_VEL
LIN {X 0,Y 291.367,Z 548.185,A -85,B 0,C 180,E1 -16527.95,E2 -16527.95} C_VEL
LIN {X 0,Y 291.377,Z 548.186,A -85,B 0,C 180,E1 -16531.158,E2 -16531.158} C_VEL
LIN {X 0,Y 291.411,Z 548.184,A -85,B 0,C 180,E1 -16534.271,E2 -16534.271} C_VEL
LIN {X 0,Y 291.375,Z 548.179,A -85,B 0,C 180,E1 -16537.299,E2 -16537.299} C_VEL
LIN {X 0,Y 291.451,Z 548.178,A -85,B 0,C 180,E1 -16540.27,E2 -16540.27} C_VEL
LIN {X 0,Y 291.548,Z 548.157,A -85,B 0,C 180,E1 -16544.623,E2 -16544.623} C_VEL
LIN {X 0,Y 291.53,Z 548.163,A -85,B 0,C 180,E1 -16548.88,E2 -16548.88} C_VEL
LIN {X 0,Y 291.702,Z 548.141,A -85,B 0,C 180,E1 -16551.688,E2 -16551.688} C_VEL
LIN {X 0,Y 291.625,Z 548.156,A -85,B 0,C 180,E1 -16554.468,E2 -16554.468} C_VEL
LIN {X 0,Y 291.884,Z 548.12,A -85,B 0,C 180,E1 -16558.62,E2 -16558.62} C_VEL
LIN {X 0,Y 291.884,Z 548.125,A -85,B 0,C 180,E1 -16561.38,E2 -16561.38} C_VEL
LIN {X 0,Y 291.74,Z 548.143,A -85,B 0,C 180,E1 -16566.918,E2 -16566.918} C_VEL
LIN {X 0,Y 291.622,Z 548.145,A -85,B 0,C 180,E1 -16569.712,E2 -16569.712} C_VEL
LIN {X 0,Y 291.516,Z 548.17,A -85,B 0,C 180,E1 -16573.951,E2 -16573.951} C_VEL
LIN {X 0,Y 291.48,Z 548.165,A -85,B 0,C 180,E1 -16576.818,E2 -16576.818} C_VEL
LIN {X 0,Y 291.444,Z 548.179,A -85,B 0,C 180,E1 -16579.875,E2 -16579.875} C_VEL
LIN {X 0,Y 291.393,Z 548.188,A -85,B 0,C 180,E1 -16584.206,E2 -16584.206} C_VEL
LIN {X 0,Y 291.408,Z 548.177,A -85,B 0,C 180,E1 -16587.273,E2 -16587.273} C_VEL
LIN {X 0,Y 291.328,Z 548.19,A -85,B 0,C 180,E1 -16590.438,E2 -16590.438} C_VEL
LIN {X 0,Y 291.339,Z 548.193,A -85,B 0,C 180,E1 -16593.699,E2 -16593.699} C_VEL
LIN {X 0,Y 291.37,Z 548.167,A -85,B 0,C 180,E1 -16597.255,E2 -16597.255} C_VEL
LIN {X 0,Y 291.365,Z 548.189,A -85,B 0,C 180,E1 -16600.637,E2 -16600.637} C_VEL
LIN {X 0,Y 291.338,Z 548.195,A -85,B 0,C 180,E1 -16604.393,E2 -16604.393} C_VEL
LIN {X 0,Y 291.384,Z 548.187,A -85,B 0,C 180,E1 -16608.392,E2 -16608.392} C_VEL
LIN {X 0,Y 291.378,Z 548.16,A -85,B 0,C 180,E1 -16611.164,E2 -16611.164} C_VEL
LIN {X 0,Y 291.382,Z 548.187,A -85,B 0,C 180,E1 -16614.631,E2 -16614.631} C_VEL
LIN {X 0,Y 291.396,Z 548.295,A -85,B 0,C 180,E1 -16615.219,E2 -16615.219} C_VEL
LIN {X 0,Y 293.507,Z 557.422,A -85,B 0,C 180,E1 -16618.547,E2 -16618.547} C_VEL
LIN {X 0,Y 295.723,Z 567.833,A -85,B 0,C 180,E1 -16622.07,E2 -16622.07} C_VEL
LIN {X 0,Y 295.98,Z 569.048,A -85,B 0,C 180,E1 -16622.373,E2 -16622.373} C_VEL
LIN {X 0,Y 299.033,Z 577.375,A -85,B 0,C 180,E1 -16622.934,E2 -16622.934} C_VEL
LIN {X 0,Y 303.917,Z 605.994,A -85,B 0,C 180,E1 -16624.137,E2 -16624.137} C_VEL
LIN {X 0,Y 304.808,Z 613.173,A -85,B 0,C 180,E1 -16624.402,E2 -16624.402} C_VEL
LIN {X 0,Y 303.122,Z 677.31,A -85,B 0,C 180,E1 -16625.927,E2 -16625.927} C_VEL
LIN {X 0,Y 302.095,Z 691.226,A -85,B 0,C 180,E1 -16626.523,E2 -16626.523} C_VEL
LIN {X 0,Y 300.85,Z 703.684,A -85,B 0,C 180,E1 -16627.33,E2 -16627.33} C_VEL
LIN {X 0,Y 299.469,Z 714.803,A -85,B 0,C 180,E1 -16628.309,E2 -16628.309} C_VEL
LIN {X 0,Y 297.772,Z 726.376,A -85,B 0,C 180,E1 -16629.629,E2 -16629.629} C_VEL
LIN {X 0,Y 296.053,Z 736.798,A -85,B 0,C 180,E1 -16631.13,E2 -16631.13} C_VEL
LIN {X 0,Y 294.574,Z 746.068,A -85,B 0,C 180,E1 -16632.804,E2 -16632.804} C_VEL
LIN {X 0,Y 293.035,Z 754.572,A -85,B 0,C 180,E1 -16634.705,E2 -16634.705} C_VEL
LIN {X 0,Y 291.654,Z 762.004,A -85,B 0,C 180,E1 -16636.768,E2 -16636.768} C_VEL
LIN {X 0,Y 290.722,Z 767.975,A -85,B 0,C 180,E1 -16638.85,E2 -16638.85} C_VEL
LIN {X 0,Y 290.048,Z 772.697,A -85,B 0,C 180,E1 -16640.94,E2 -16640.94} C_VEL
LIN {X 0,Y 289.607,Z 776.309,A -85,B 0,C 180,E1 -16643.032,E2 -16643.032} C_VEL
LIN {X 0,Y 289.478,Z 778.259,A -85,B 0,C 180,E1 -16644.507,E2 -16644.507} C_VEL
LIN {X 0,Y 289.438,Z 780.567,A -85,B 0,C 180,E1 -16647.218,E2 -16647.218} C_VEL
LIN {X 0,Y 289.405,Z 782.093,A -85,B 0,C 180,E1 -16650.001,E2 -16650.001} C_VEL
LIN {X 0,Y 289.389,Z 783.299,A -85,B 0,C 180,E1 -16651.393,E2 -16651.393} C_VEL
LIN {X 0,Y 289.449,Z 783.929,A -85,B 0,C 180,E1 -16652.785,E2 -16652.785} C_VEL
LIN {X 0,Y 289.497,Z 783.98,A -85,B 0,C 180,E1 -16654.178,E2 -16654.178} C_VEL
LIN {X 0,Y 289.712,Z 783.174,A -85,B 0,C 180,E1 -16655.955,E2 -16655.955} C_VEL
LIN {X 0,Y 289.873,Z 782.356,A -85,B 0,C 180,E1 -16656.964,E2 -16656.964} C_VEL
LIN {X 0,Y 290.459,Z 779.467,A -85,B 0,C 180,E1 -16659.05,E2 -16659.05} C_VEL
LIN {X 0,Y 291.301,Z 775.248,A -85,B 0,C 180,E1 -16661.13,E2 -16661.13} C_VEL
LIN {X 0,Y 292.358,Z 769.363,A -85,B 0,C 180,E1 -16663.202,E2 -16663.202} C_VEL
LIN {X 0,Y 293.514,Z 762.942,A -85,B 0,C 180,E1 -16664.917,E2 -16664.917} C_VEL
LIN {X 0,Y 294.819,Z 754.981,A -85,B 0,C 180,E1 -16666.623,E2 -16666.623} C_VEL
LIN {X 0,Y 295.887,Z 746.918,A -85,B 0,C 180,E1 -16667.987,E2 -16667.987} C_VEL
LIN {X 0,Y 296.772,Z 738.443,A -85,B 0,C 180,E1 -16669.166,E2 -16669.166} C_VEL
LIN {X 0,Y 297.802,Z 727.325,A -85,B 0,C 180,E1 -16670.372,E2 -16670.372} C_VEL
LIN {X 0,Y 298.378,Z 722.18,A -85,B 0,C 180,E1 -16670.871,E2 -16670.871} C_VEL
LIN {X 0,Y 299.926,Z 711.111,A -85,B 0,C 180,E1 -16672.02,E2 -16672.02} C_VEL
LIN {X 0,Y 301.348,Z 698.844,A -85,B 0,C 180,E1 -16672.996,E2 -16672.996} C_VEL
LIN {X 0,Y 302.468,Z 686.842,A -85,B 0,C 180,E1 -16673.675,E2 -16673.675} C_VEL
LIN {X 0,Y 303.211,Z 673.659,A -85,B 0,C 180,E1 -16674.159,E2 -16674.159} C_VEL
LIN {X 0,Y 304.303,Z 634.445,A -85,B 0,C 180,E1 -16675.112,E2 -16675.112} C_VEL
LIN {X 0,Y 304.599,Z 631.291,A -85,B 0,C 180,E1 -16675.269,E2 -16675.269} C_VEL
LIN {X 0,Y 309.005,Z 614.824,A -85,B 0,C 180,E1 -16676.675,E2 -16676.675} C_VEL
LIN {X 0,Y 311.652,Z 599.909,A -85,B 0,C 180,E1 -16678.513,E2 -16678.513} C_VEL
LIN {X 0,Y 312.12,Z 595.029,A -85,B 0,C 180,E1 -16679.315,E2 -16679.315} C_VEL
LIN {X 0,Y 311.744,Z 590.793,A -85,B 0,C 180,E1 -16680.327,E2 -16680.327} C_VEL
LIN {X 0,Y 311.012,Z 583.478,A -85,B 0,C 180,E1 -16682.435,E2 -16682.435} C_VEL
LIN {X 0,Y 310.672,Z 581.458,A -85,B 0,C 180,E1 -16683.174,E2 -16683.174} C_VEL
LIN {X 0,Y 309.098,Z 578.621,A -85,B 0,C 180,E1 -16685.061,E2 -16685.061} C_VEL
LIN {X 0,Y 307.813,Z 576.693,A -85,B 0,C 180,E1 -16686.953,E2 -16686.953} C_VEL
LIN {X 0,Y 306.461,Z 575.22,A -85,B 0,C 180,E1 -16689.951,E2 -16689.951} C_VEL
LIN {X 0,Y 306.198,Z 575.202,A -85,B 0,C 180,E1 -16692.737,E2 -16692.737} C_VEL
LIN {X 0,Y 306.512,Z 576.436,A -85,B 0,C 180,E1 -16695.301,E2 -16695.301} C_VEL
LIN {X 0,Y 307.357,Z 579.712,A -85,B 0,C 180,E1 -16698.462,E2 -16698.462} C_VEL
LIN {X 0,Y 308.587,Z 584.336,A -85,B 0,C 180,E1 -16701.352,E2 -16701.352} C_VEL
LIN {X 0,Y 309.675,Z 589.652,A -85,B 0,C 180,E1 -16703.838,E2 -16703.838} C_VEL
LIN {X 0,Y 310.639,Z 596.368,A -85,B 0,C 180,E1 -16706.359,E2 -16706.359} C_VEL
LIN {X 0,Y 310.838,Z 598.712,A -85,B 0,C 180,E1 -16707.137,E2 -16707.137} C_VEL
LIN {X 0,Y 310.424,Z 601.443,A -85,B 0,C 180,E1 -16707.829,E2 -16707.829} C_VEL
LIN {X 0,Y 305.722,Z 623.029,A -85,B 0,C 180,E1 -16712.628,E2 -16712.628} C_VEL
LIN {X 0,Y 304.028,Z 632.47,A -85,B 0,C 180,E1 -16714.65,E2 -16714.65} C_VEL
LIN {X 0,Y 306.521,Z 646.023,A -85,B 0,C 180,E1 -16715.961,E2 -16715.961} C_VEL
LIN {X 0,Y 308.268,Z 659.87,A -85,B 0,C 180,E1 -16717.041,E2 -16717.041} C_VEL
LIN {X 0,Y 308.259,Z 663.504,A -85,B 0,C 180,E1 -16717.241,E2 -16717.241} C_VEL
LIN {X 0,Y 304.698,Z 707.235,A -85,B 0,C 180,E1 -16719.008,E2 -16719.008} C_VEL
LIN {X 0,Y 303.455,Z 718.214,A -85,B 0,C 180,E1 -16719.672,E2 -16719.672} C_VEL
LIN {X 0,Y 301.819,Z 729.244,A -85,B 0,C 180,E1 -16720.621,E2 -16720.621} C_VEL
LIN {X 0,Y 300.099,Z 739.165,A -85,B 0,C 180,E1 -16721.746,E2 -16721.746} C_VEL
LIN {X 0,Y 298.526,Z 747.088,A -85,B 0,C 180,E1 -16722.886,E2 -16722.886} C_VEL
LIN {X 0,Y 296.915,Z 754.386,A -85,B 0,C 180,E1 -16724.204,E2 -16724.204} C_VEL
LIN {X 0,Y 295.419,Z 760.419,A -85,B 0,C 180,E1 -16725.535,E2 -16725.535} C_VEL
LIN {X 0,Y 293.79,Z 766.556,A -85,B 0,C 180,E1 -16727.216,E2 -16727.216} C_VEL
LIN {X 0,Y 292.524,Z 771.304,A -85,B 0,C 180,E1 -16728.919,E2 -16728.919} C_VEL
LIN {X 0,Y 291.681,Z 774.296,A -85,B 0,C 180,E1 -16730.29,E2 -16730.29} C_VEL
LIN {X 0,Y 290.781,Z 777.369,A -85,B 0,C 180,E1 -16732.29,E2 -16732.29} C_VEL
LIN {X 0,Y 290.542,Z 778.269,A -85,B 0,C 180,E1 -16733.053,E2 -16733.053} C_VEL
LIN {X 0,Y 290.07,Z 779.333,A -85,B 0,C 180,E1 -16734.439,E2 -16734.439} C_VEL
LIN {X 0,Y 289.709,Z 779.824,A -85,B 0,C 180,E1 -16735.827,E2 -16735.827} C_VEL
LIN {X 0,Y 289.529,Z 779.745,A -85,B 0,C 180,E1 -16737.217,E2 -16737.217} C_VEL
LIN {X 0,Y 289.397,Z 779.089,A -85,B 0,C 180,E1 -16738.609,E2 -16738.609} C_VEL
LIN {X 0,Y 289.373,Z 777.844,A -85,B 0,C 180,E1 -16740,E2 -16740} C_VEL
LIN {X 0,Y 289.427,Z 774.783,A -85,B 0,C 180,E1 -16742.087,E2 -16742.087} C_VEL
LIN {X 0,Y 289.64,Z 770.236,A -85,B 0,C 180,E1 -16744.175,E2 -16744.175} C_VEL
LIN {X 0,Y 289.752,Z 764.617,A -85,B 0,C 180,E1 -16746.024,E2 -16746.024} C_VEL
LIN {X 0,Y 290.139,Z 758.217,A -85,B 0,C 180,E1 -16747.688,E2 -16747.688} C_VEL
LIN {X 0,Y 290.572,Z 749.692,A -85,B 0,C 180,E1 -16749.396,E2 -16749.396} C_VEL
LIN {X 0,Y 290.914,Z 742.056,A -85,B 0,C 180,E1 -16750.615,E2 -16750.615} C_VEL
LIN {X 0,Y 291.527,Z 732.662,A -85,B 0,C 180,E1 -16751.825,E2 -16751.825} C_VEL
LIN {X 0,Y 291.994,Z 722.887,A -85,B 0,C 180,E1 -16752.776,E2 -16752.776} C_VEL
LIN {X 0,Y 292.381,Z 712.365,A -85,B 0,C 180,E1 -16753.554,E2 -16753.554} C_VEL
LIN {X 0,Y 292.748,Z 699.991,A -85,B 0,C 180,E1 -16754.157,E2 -16754.157} C_VEL
LIN {X 0,Y 293.74,Z 653.578,A -85,B 0,C 180,E1 -16755.837,E2 -16755.837} C_VEL
LIN {X 0,Y 292.243,Z 632.193,A -85,B 0,C 180,E1 -16756.674,E2 -16756.674} C_VEL
LIN {X 0,Y 293.184,Z 617.219,A -85,B 0,C 180,E1 -16759.609,E2 -16759.609} C_VEL
LIN {X 0,Y 294.488,Z 599.251,A -85,B 0,C 180,E1 -16763.19,E2 -16763.19} C_VEL
LIN {X 0,Y 296.239,Z 577.336,A -85,B 0,C 180,E1 -16767.556,E2 -16767.556} C_VEL
LIN {X 0,Y 296.578,Z 573.647,A -85,B 0,C 180,E1 -16768.29,E2 -16768.29} C_VEL
LIN {X 0,Y 294.632,Z 563.267,A -85,B 0,C 180,E1 -16770.511,E2 -16770.511} C_VEL
LIN {X 0,Y 291.435,Z 548.342,A -85,B 0,C 180,E1 -16773.838,E2 -16773.838} C_VEL
LIN {X 0,Y 291.386,Z 548.189,A -85,B 0,C 180,E1 -16777.255,E2 -16777.255} C_VEL
LIN {X 0,Y 291.339,Z 548.171,A -85,B 0,C 180,E1 -16780.642,E2 -16780.642} C_VEL
LIN {X 0,Y 291.318,Z 548.162,A -85,B 0,C 180,E1 -16784.397,E2 -16784.397} C_VEL
LIN {X 0,Y 291.359,Z 548.179,A -85,B 0,C 180,E1 -16788.397,E2 -16788.397} C_VEL
LIN {X 0,Y 291.352,Z 548.163,A -85,B 0,C 180,E1 -16791.157,E2 -16791.157} C_VEL
LIN {X 0,Y 291.365,Z 548.182,A -85,B 0,C 180,E1 -16794.625,E2 -16794.625} C_VEL
LIN {X 0,Y 291.377,Z 548.186,A -85,B 0,C 180,E1 -16797.95,E2 -16797.95} C_VEL
LIN {X 0,Y 291.407,Z 548.29,A -85,B 0,C 180,E1 -16799.771,E2 -16799.771} C_VEL
LIN {X 0,Y 292.817,Z 554.338,A -85,B 0,C 180,E1 -16802.106,E2 -16802.106} C_VEL
LIN {X 0,Y 295.4,Z 560.275,A -85,B 0,C 180,E1 -16802.597,E2 -16802.597} C_VEL
LIN {X 0,Y 302.449,Z 577.318,A -85,B 0,C 180,E1 -16803.738,E2 -16803.738} C_VEL
LIN {X 0,Y 304.393,Z 583.287,A -85,B 0,C 180,E1 -16804.074,E2 -16804.074} C_VEL
LIN {X 0,Y 305.379,Z 588.431,A -85,B 0,C 180,E1 -16804.296,E2 -16804.296} C_VEL
LIN {X 0,Y 303.386,Z 660.637,A -85,B 0,C 180,E1 -16805.992,E2 -16805.992} C_VEL
LIN {X 0,Y 302.572,Z 674.022,A -85,B 0,C 180,E1 -16806.56,E2 -16806.56} C_VEL
LIN {X 0,Y 301.547,Z 686.775,A -85,B 0,C 180,E1 -16807.383,E2 -16807.383} C_VEL
LIN {X 0,Y 300.236,Z 698.092,A -85,B 0,C 180,E1 -16808.365,E2 -16808.365} C_VEL
LIN {X 0,Y 298.608,Z 709.736,A -85,B 0,C 180,E1 -16809.686,E2 -16809.686} C_VEL
LIN {X 0,Y 297.184,Z 719.436,A -85,B 0,C 180,E1 -16811.076,E2 -16811.076} C_VEL
LIN {X 0,Y 295.701,Z 728.721,A -85,B 0,C 180,E1 -16812.716,E2 -16812.716} C_VEL
LIN {X 0,Y 294.22,Z 736.588,A -85,B 0,C 180,E1 -16814.41,E2 -16814.41} C_VEL
LIN {X 0,Y 292.812,Z 744.27,A -85,B 0,C 180,E1 -16816.465,E2 -16816.465} C_VEL
LIN {X 0,Y 291.474,Z 751.325,A -85,B 0,C 180,E1 -16818.877,E2 -16818.877} C_VEL
LIN {X 0,Y 290.624,Z 756.021,A -85,B 0,C 180,E1 -16820.955,E2 -16820.955} C_VEL
LIN {X 0,Y 290.035,Z 760.229,A -85,B 0,C 180,E1 -16823.463,E2 -16823.463} C_VEL
LIN {X 0,Y 289.706,Z 762.856,A -85,B 0,C 180,E1 -16825.825,E2 -16825.825} C_VEL
LIN {X 0,Y 289.457,Z 764.463,A -85,B 0,C 180,E1 -16828.607,E2 -16828.607} C_VEL
LIN {X 0,Y 289.444,Z 764.694,A -85,B 0,C 180,E1 -16829.999,E2 -16829.999} C_VEL
LIN {X 0,Y 289.457,Z 764.503,A -85,B 0,C 180,E1 -16831.39,E2 -16831.39} C_VEL
LIN {X 0,Y 289.701,Z 762.951,A -85,B 0,C 180,E1 -16834.172,E2 -16834.172} C_VEL
LIN {X 0,Y 290.014,Z 760.422,A -85,B 0,C 180,E1 -16836.5,E2 -16836.5} C_VEL
LIN {X 0,Y 290.62,Z 756.253,A -85,B 0,C 180,E1 -16839.042,E2 -16839.042} C_VEL
LIN {X 0,Y 291.443,Z 751.621,A -85,B 0,C 180,E1 -16841.122,E2 -16841.122} C_VEL
LIN {X 0,Y 292.717,Z 744.638,A -85,B 0,C 180,E1 -16843.537,E2 -16843.537} C_VEL
LIN {X 0,Y 294.146,Z 737.064,A -85,B 0,C 180,E1 -16845.591,E2 -16845.591} C_VEL
LIN {X 0,Y 295.999,Z 727.527,A -85,B 0,C 180,E1 -16847.62,E2 -16847.62} C_VEL
LIN {X 0,Y 297.483,Z 717.687,A -85,B 0,C 180,E1 -16849.313,E2 -16849.313} C_VEL
LIN {X 0,Y 298.919,Z 708.001,A -85,B 0,C 180,E1 -16850.649,E2 -16850.649} C_VEL
LIN {X 0,Y 300.391,Z 697.505,A -85,B 0,C 180,E1 -16851.801,E2 -16851.801} C_VEL
LIN {X 0,Y 301.689,Z 685.98,A -85,B 0,C 180,E1 -16852.784,E2 -16852.784} C_VEL
LIN {X 0,Y 302.72,Z 672.948,A -85,B 0,C 180,E1 -16853.607,E2 -16853.607} C_VEL
LIN {X 0,Y 303.529,Z 660.1,A -85,B 0,C 180,E1 -16854.129,E2 -16854.129} C_VEL
LIN {X 0,Y 305.349,Z 588.192,A -85,B 0,C 180,E1 -16855.828,E2 -16855.828} C_VEL
LIN {X 0,Y 303.671,Z 580.478,A -85,B 0,C 180,E1 -16856.182,E2 -16856.182} C_VEL
LIN {X 0,Y 296.337,Z 562.404,A -85,B 0,C 180,E1 -16857.37,E2 -16857.37} C_VEL
LIN {X 0,Y 292.832,Z 554.452,A -85,B 0,C 180,E1 -16857.994,E2 -16857.994} C_VEL
LIN {X 0,Y 291.441,Z 548.492,A -85,B 0,C 180,E1 -16860.225,E2 -16860.225} C_VEL
LIN {X 0,Y 291.384,Z 548.208,A -85,B 0,C 180,E1 -16860.43,E2 -16860.43} C_VEL
LIN {X 0,Y 291.387,Z 548.187,A -85,B 0,C 180,E1 -16864.91,E2 -16864.91} C_VEL
LIN {X 0,Y 291.396,Z 548.186,A -85,B 0,C 180,E1 -16867.259,E2 -16867.259} C_VEL
LIN {X 0,Y 291.335,Z 548.183,A -85,B 0,C 180,E1 -16870.322,E2 -16870.322} C_VEL
LIN {X 0,Y 290.659,Z 548.279,A -85,B 0,C 180,E1 -16871.476,E2 -16871.476} C_VEL
LIN {X 0,Y 287.814,Z 548.626,A -85,B 0,C 180,E1 -16873.355,E2 -16873.355} C_VEL
LIN {X 0,Y 285.397,Z 548.924,A -85,B 0,C 180,E1 -16874.881,E2 -16874.881} C_VEL
LIN {X 0,Y 284.348,Z 549.054,A -85,B 0,C 180,E1 -16876.062,E2 -16876.062} C_VEL
LIN {X 0,Y 284.256,Z 549.065,A -85,B 0,C 180,E1 -16876.463,E2 -16876.463} C_VEL
LIN {X 0,Y 284.346,Z 549.048,A -85,B 0,C 180,E1 -16880.012,E2 -16880.012} C_VEL
LIN {X 0,Y 284.348,Z 549.055,A -85,B 0,C 180,E1 -16883.616,E2 -16883.616} C_VEL
LIN {X 0,Y 284.303,Z 549.065,A -85,B 0,C 180,E1 -16887.188,E2 -16887.188} C_VEL
LIN {X 0,Y 284.353,Z 549.063,A -85,B 0,C 180,E1 -16890.375,E2 -16890.375} C_VEL
LIN {X 0,Y 284.372,Z 549.056,A -85,B 0,C 180,E1 -16893.586,E2 -16893.586} C_VEL
LIN {X 0,Y 284.36,Z 549.058,A -85,B 0,C 180,E1 -16896.706,E2 -16896.706} C_VEL
LIN {X 0,Y 284.397,Z 549.06,A -85,B 0,C 180,E1 -16901.261,E2 -16901.261} C_VEL
LIN {X 0,Y 284.485,Z 549.036,A -85,B 0,C 180,E1 -16904.459,E2 -16904.459} C_VEL
LIN {X 0,Y 284.481,Z 549.042,A -85,B 0,C 180,E1 -16908.601,E2 -16908.601} C_VEL
LIN {X 0,Y 284.652,Z 549.017,A -85,B 0,C 180,E1 -16911.481,E2 -16911.481} C_VEL
LIN {X 0,Y 284.595,Z 549.032,A -85,B 0,C 180,E1 -16914.331,E2 -16914.331} C_VEL
LIN {X 0,Y 284.85,Z 548.997,A -85,B 0,C 180,E1 -16918.586,E2 -16918.586} C_VEL
LIN {X 0,Y 284.85,Z 549,A -85,B 0,C 180,E1 -16921.414,E2 -16921.414} C_VEL
LIN {X 0,Y 284.692,Z 549.022,A -85,B 0,C 180,E1 -16927.09,E2 -16927.09} C_VEL
LIN {X 0,Y 284.56,Z 549.024,A -85,B 0,C 180,E1 -16929.956,E2 -16929.956} C_VEL
LIN {X 0,Y 284.475,Z 549.045,A -85,B 0,C 180,E1 -16934.303,E2 -16934.303} C_VEL
LIN {X 0,Y 284.419,Z 549.047,A -85,B 0,C 180,E1 -16937.249,E2 -16937.249} C_VEL
LIN {X 0,Y 284.372,Z 549.058,A -85,B 0,C 180,E1 -16940.243,E2 -16940.243} C_VEL
LIN {X 0,Y 284.362,Z 549.066,A -85,B 0,C 180,E1 -16943.876,E2 -16943.876} C_VEL
LIN {X 0,Y 284.385,Z 549.051,A -85,B 0,C 180,E1 -16947.172,E2 -16947.172} C_VEL
LIN {X 0,Y 284.288,Z 549.066,A -85,B 0,C 180,E1 -16951.275,E2 -16951.275} C_VEL
LIN {X 0,Y 284.335,Z 549.048,A -85,B 0,C 180,E1 -16955.349,E2 -16955.349} C_VEL
LIN {X 0,Y 284.307,Z 549.057,A -85,B 0,C 180,E1 -16958.17,E2 -16958.17} C_VEL
LIN {X 0,Y 284.292,Z 549.055,A -85,B 0,C 180,E1 -16962.132,E2 -16962.132} C_VEL
LIN {X 0,Y 284.313,Z 549.061,A -85,B 0,C 180,E1 -16966.203,E2 -16966.203} C_VEL
LIN {X 0,Y 284.347,Z 549.055,A -85,B 0,C 180,E1 -16970.014,E2 -16970.014} C_VEL
LIN {X 0,Y 284.336,Z 549.053,A -85,B 0,C 180,E1 -16974.198,E2 -16974.198} C_VEL
LIN {X 0,Y 284.373,Z 549.32,A -85,B 0,C 180,E1 -16974.713,E2 -16974.713} C_VEL
LIN {X 0,Y 286.568,Z 558.667,A -85,B 0,C 180,E1 -16978.181,E2 -16978.181} C_VEL
LIN {X 0,Y 288.658,Z 568.548,A -85,B 0,C 180,E1 -16981.573,E2 -16981.573} C_VEL
LIN {X 0,Y 290.758,Z 574.021,A -85,B 0,C 180,E1 -16982.013,E2 -16982.013} C_VEL
LIN {X 0,Y 292.982,Z 579.885,A -85,B 0,C 180,E1 -16982.401,E2 -16982.401} C_VEL
LIN {X 0,Y 297.652,Z 607.907,A -85,B 0,C 180,E1 -16983.607,E2 -16983.607} C_VEL
LIN {X 0,Y 298.383,Z 614.434,A -85,B 0,C 180,E1 -16983.847,E2 -16983.847} C_VEL
LIN {X 0,Y 296.668,Z 677.119,A -85,B 0,C 180,E1 -16985.369,E2 -16985.369} C_VEL
LIN {X 0,Y 295.683,Z 690.269,A -85,B 0,C 180,E1 -16985.936,E2 -16985.936} C_VEL
LIN {X 0,Y 294.424,Z 702.372,A -85,B 0,C 180,E1 -16986.714,E2 -16986.714} C_VEL
LIN {X 0,Y 292.89,Z 714.603,A -85,B 0,C 180,E1 -16987.796,E2 -16987.796} C_VEL
LIN {X 0,Y 291.111,Z 726.175,A -85,B 0,C 180,E1 -16989.141,E2 -16989.141} C_VEL
LIN {X 0,Y 289.321,Z 736.596,A -85,B 0,C 180,E1 -16990.674,E2 -16990.674} C_VEL
LIN {X 0,Y 287.867,Z 744.984,A -85,B 0,C 180,E1 -16992.204,E2 -16992.204} C_VEL
LIN {X 0,Y 286.405,Z 752.992,A -85,B 0,C 180,E1 -16993.976,E2 -16993.976} C_VEL
LIN {X 0,Y 284.968,Z 760.679,A -85,B 0,C 180,E1 -16996.088,E2 -16996.088} C_VEL
LIN {X 0,Y 284.001,Z 765.948,A -85,B 0,C 180,E1 -16997.859,E2 -16997.859} C_VEL
LIN {X 0,Y 283.2,Z 771.056,A -85,B 0,C 180,E1 -16999.997,E2 -16999.997} C_VEL
LIN {X 0,Y 282.684,Z 775.03,A -85,B 0,C 180,E1 -17002.142,E2 -17002.142} C_VEL
LIN {X 0,Y 282.37,Z 778.301,A -85,B 0,C 180,E1 -17004.609,E2 -17004.609} C_VEL
LIN {X 0,Y 282.346,Z 780.362,A -85,B 0,C 180,E1 -17007.148,E2 -17007.148} C_VEL
LIN {X 0,Y 282.326,Z 781.624,A -85,B 0,C 180,E1 -17010.001,E2 -17010.001} C_VEL
LIN {X 0,Y 282.314,Z 782.983,A -85,B 0,C 180,E1 -17011.428,E2 -17011.428} C_VEL
LIN {X 0,Y 282.359,Z 783.781,A -85,B 0,C 180,E1 -17012.855,E2 -17012.855} C_VEL
LIN {X 0,Y 282.409,Z 784,A -85,B 0,C 180,E1 -17014.283,E2 -17014.283} C_VEL
LIN {X 0,Y 282.595,Z 783.533,A -85,B 0,C 180,E1 -17015.855,E2 -17015.855} C_VEL
LIN {X 0,Y 282.832,Z 782.61,A -85,B 0,C 180,E1 -17017.138,E2 -17017.138} C_VEL
LIN {X 0,Y 283.476,Z 780.039,A -85,B 0,C 180,E1 -17019.275,E2 -17019.275} C_VEL
LIN {X 0,Y 284.082,Z 777.569,A -85,B 0,C 180,E1 -17020.694,E2 -17020.694} C_VEL
LIN {X 0,Y 284.747,Z 774.413,A -85,B 0,C 180,E1 -17022.111,E2 -17022.111} C_VEL
LIN {X 0,Y 285.711,Z 769.404,A -85,B 0,C 180,E1 -17023.878,E2 -17023.878} C_VEL
LIN {X 0,Y 287.132,Z 763.062,A -85,B 0,C 180,E1 -17025.62,E2 -17025.62} C_VEL
LIN {X 0,Y 288.464,Z 755.736,A -85,B 0,C 180,E1 -17027.249,E2 -17027.249} C_VEL
LIN {X 0,Y 289.944,Z 746.032,A -85,B 0,C 180,E1 -17028.927,E2 -17028.927} C_VEL
LIN {X 0,Y 290.841,Z 738.809,A -85,B 0,C 180,E1 -17029.959,E2 -17029.959} C_VEL
LIN {X 0,Y 292.028,Z 728.189,A -85,B 0,C 180,E1 -17031.162,E2 -17031.162} C_VEL
LIN {X 0,Y 292.87,Z 716.951,A -85,B 0,C 180,E1 -17032.115,E2 -17032.115} C_VEL
LIN {X 0,Y 293.362,Z 710.907,A -85,B 0,C 180,E1 -17032.54,E2 -17032.54} C_VEL
LIN {X 0,Y 294.832,Z 698.636,A -85,B 0,C 180,E1 -17033.534,E2 -17033.534} C_VEL
LIN {X 0,Y 296.054,Z 685.725,A -85,B 0,C 180,E1 -17034.268,E2 -17034.268} C_VEL
LIN {X 0,Y 296.796,Z 671.962,A -85,B 0,C 180,E1 -17034.762,E2 -17034.762} C_VEL
LIN {X 0,Y 297.332,Z 655.597,A -85,B 0,C 180,E1 -17035.181,E2 -17035.181} C_VEL
LIN {X 0,Y 299.782,Z 631.573,A -85,B 0,C 180,E1 -17036.265,E2 -17036.265} C_VEL
LIN {X 0,Y 304.401,Z 615.039,A -85,B 0,C 180,E1 -17037.753,E2 -17037.753} C_VEL
LIN {X 0,Y 307.193,Z 600.87,A -85,B 0,C 180,E1 -17039.614,E2 -17039.614} C_VEL
LIN {X 0,Y 307.336,Z 597.85,A -85,B 0,C 180,E1 -17040.205,E2 -17040.205} C_VEL
LIN {X 0,Y 306.765,Z 591.143,A -85,B 0,C 180,E1 -17042.04,E2 -17042.04} C_VEL
LIN {X 0,Y 306.396,Z 587.042,A -85,B 0,C 180,E1 -17043.403,E2 -17043.403} C_VEL
LIN {X 0,Y 304.95,Z 584.349,A -85,B 0,C 180,E1 -17045.182,E2 -17045.182} C_VEL
LIN {X 0,Y 303.133,Z 581.78,A -85,B 0,C 180,E1 -17047.975,E2 -17047.975} C_VEL
LIN {X 0,Y 302.153,Z 580.836,A -85,B 0,C 180,E1 -17050.639,E2 -17050.639} C_VEL
LIN {X 0,Y 301.909,Z 580.815,A -85,B 0,C 180,E1 -17052.461,E2 -17052.461} C_VEL
LIN {X 0,Y 301.982,Z 581.411,A -85,B 0,C 180,E1 -17054.283,E2 -17054.283} C_VEL
LIN {X 0,Y 302.164,Z 582.743,A -85,B 0,C 180,E1 -17056.14,E2 -17056.14} C_VEL
LIN {X 0,Y 302.908,Z 585.978,A -85,B 0,C 180,E1 -17059.028,E2 -17059.028} C_VEL
LIN {X 0,Y 303.921,Z 590.635,A -85,B 0,C 180,E1 -17061.836,E2 -17061.836} C_VEL
LIN {X 0,Y 304.805,Z 596.151,A -85,B 0,C 180,E1 -17064.336,E2 -17064.336} C_VEL
LIN {X 0,Y 305.345,Z 601.885,A -85,B 0,C 180,E1 -17066.468,E2 -17066.468} C_VEL
LIN {X 0,Y 305.084,Z 604.247,A -85,B 0,C 180,E1 -17067.134,E2 -17067.134} C_VEL
LIN {X 0,Y 300.31,Z 624.337,A -85,B 0,C 180,E1 -17071.712,E2 -17071.712} C_VEL
LIN {X 0,Y 298.668,Z 632.801,A -85,B 0,C 180,E1 -17073.557,E2 -17073.557} C_VEL
LIN {X 0,Y 301.277,Z 647.597,A -85,B 0,C 180,E1 -17075.06,E2 -17075.06} C_VEL
LIN {X 0,Y 302.78,Z 659.677,A -85,B 0,C 180,E1 -17076.076,E2 -17076.076} C_VEL
LIN {X 0,Y 302.979,Z 663.992,A -85,B 0,C 180,E1 -17076.359,E2 -17076.359} C_VEL
LIN {X 0,Y 299.08,Z 707.522,A -85,B 0,C 180,E1 -17078.187,E2 -17078.187} C_VEL
LIN {X 0,Y 297.698,Z 718.952,A -85,B 0,C 180,E1 -17078.899,E2 -17078.899} C_VEL
LIN {X 0,Y 295.966,Z 729.784,A -85,B 0,C 180,E1 -17079.86,E2 -17079.86} C_VEL
LIN {X 0,Y 294.129,Z 739.611,A -85,B 0,C 180,E1 -17081,E2 -17081} C_VEL
LIN {X 0,Y 292.395,Z 747.375,A -85,B 0,C 180,E1 -17082.154,E2 -17082.154} C_VEL
LIN {X 0,Y 290.674,Z 754.569,A -85,B 0,C 180,E1 -17083.495,E2 -17083.495} C_VEL
LIN {X 0,Y 288.687,Z 761.974,A -85,B 0,C 180,E1 -17085.19,E2 -17085.19} C_VEL
LIN {X 0,Y 287.282,Z 766.728,A -85,B 0,C 180,E1 -17086.561,E2 -17086.561} C_VEL
LIN {X 0,Y 286.154,Z 770.593,A -85,B 0,C 180,E1 -17087.95,E2 -17087.95} C_VEL
LIN {X 0,Y 284.743,Z 774.97,A -85,B 0,C 180,E1 -17090.051,E2 -17090.051} C_VEL
LIN {X 0,Y 283.71,Z 778.04,A -85,B 0,C 180,E1 -17092.259,E2 -17092.259} C_VEL
LIN {X 0,Y 283.025,Z 779.627,A -85,B 0,C 180,E1 -17094.3,E2 -17094.3} C_VEL
LIN {X 0,Y 282.642,Z 779.972,A -85,B 0,C 180,E1 -17095.722,E2 -17095.722} C_VEL
LIN {X 0,Y 282.442,Z 779.722,A -85,B 0,C 180,E1 -17097.147,E2 -17097.147} C_VEL
LIN {X 0,Y 282.324,Z 778.906,A -85,B 0,C 180,E1 -17098.574,E2 -17098.574} C_VEL
LIN {X 0,Y 282.284,Z 776.64,A -85,B 0,C 180,E1 -17100.713,E2 -17100.713} C_VEL
LIN {X 0,Y 282.446,Z 772.798,A -85,B 0,C 180,E1 -17102.853,E2 -17102.853} C_VEL
LIN {X 0,Y 282.572,Z 768.053,A -85,B 0,C 180,E1 -17104.754,E2 -17104.754} C_VEL
LIN {X 0,Y 282.842,Z 761.326,A -85,B 0,C 180,E1 -17106.778,E2 -17106.778} C_VEL
LIN {X 0,Y 283.191,Z 755.264,A -85,B 0,C 180,E1 -17108.204,E2 -17108.204} C_VEL
LIN {X 0,Y 283.576,Z 747.856,A -85,B 0,C 180,E1 -17109.63,E2 -17109.63} C_VEL
LIN {X 0,Y 284.072,Z 738.585,A -85,B 0,C 180,E1 -17111.054,E2 -17111.054} C_VEL
LIN {X 0,Y 284.568,Z 729.693,A -85,B 0,C 180,E1 -17112.118,E2 -17112.118} C_VEL
LIN {X 0,Y 285.041,Z 719.311,A -85,B 0,C 180,E1 -17113.093,E2 -17113.093} C_VEL
LIN {X 0,Y 285.433,Z 707.796,A -85,B 0,C 180,E1 -17113.845,E2 -17113.845} C_VEL
LIN {X 0,Y 285.744,Z 695.577,A -85,B 0,C 180,E1 -17114.375,E2 -17114.375} C_VEL
LIN {X 0,Y 286.688,Z 654.024,A -85,B 0,C 180,E1 -17115.931,E2 -17115.931} C_VEL
LIN {X 0,Y 285.179,Z 632.395,A -85,B 0,C 180,E1 -17116.794,E2 -17116.794} C_VEL
LIN {X 0,Y 286.078,Z 619.352,A -85,B 0,C 180,E1 -17119.369,E2 -17119.369} C_VEL
LIN {X 0,Y 287.592,Z 597.603,A -85,B 0,C 180,E1 -17123.78,E2 -17123.78} C_VEL
LIN {X 0,Y 289.299,Z 577.368,A -85,B 0,C 180,E1 -17127.882,E2 -17127.882} C_VEL
LIN {X 0,Y 289.404,Z 573.106,A -85,B 0,C 180,E1 -17128.756,E2 -17128.756} C_VEL
LIN {X 0,Y 286.232,Z 557.981,A -85,B 0,C 180,E1 -17132.071,E2 -17132.071} C_VEL
LIN {X 0,Y 284.385,Z 549.22,A -85,B 0,C 180,E1 -17134.096,E2 -17134.096} C_VEL
LIN {X 0,Y 284.323,Z 549.07,A -85,B 0,C 180,E1 -17138.167,E2 -17138.167} C_VEL
LIN {X 0,Y 284.273,Z 549.027,A -85,B 0,C 180,E1 -17142.124,E2 -17142.124} C_VEL
LIN {X 0,Y 284.293,Z 549.068,A -85,B 0,C 180,E1 -17146.195,E2 -17146.195} C_VEL
LIN {X 0,Y 284.312,Z 549.037,A -85,B 0,C 180,E1 -17150.023,E2 -17150.023} C_VEL
LIN {X 0,Y 284.335,Z 549.068,A -85,B 0,C 180,E1 -17153.613,E2 -17153.613} C_VEL
LIN {X 0,Y 284.312,Z 549.071,A -85,B 0,C 180,E1 -17157.189,E2 -17157.189} C_VEL
LIN {X 0,Y 284.351,Z 549.185,A -85,B 0,C 180,E1 -17159.207,E2 -17159.207} C_VEL
LIN {X 0,Y 285.621,Z 554.586,A -85,B 0,C 180,E1 -17161.344,E2 -17161.344} C_VEL
LIN {X 0,Y 288.548,Z 561.056,A -85,B 0,C 180,E1 -17161.904,E2 -17161.904} C_VEL
LIN {X 0,Y 296.09,Z 579.021,A -85,B 0,C 180,E1 -17163.168,E2 -17163.168} C_VEL
LIN {X 0,Y 298.162,Z 585.124,A -85,B 0,C 180,E1 -17163.533,E2 -17163.533} C_VEL
LIN {X 0,Y 298.976,Z 589.526,A -85,B 0,C 180,E1 -17163.727,E2 -17163.727} C_VEL
LIN {X 0,Y 296.928,Z 660.859,A -85,B 0,C 180,E1 -17165.436,E2 -17165.436} C_VEL
LIN {X 0,Y 296.084,Z 674.237,A -85,B 0,C 180,E1 -17166.014,E2 -17166.014} C_VEL
LIN {X 0,Y 295.002,Z 686.988,A -85,B 0,C 180,E1 -17166.852,E2 -17166.852} C_VEL
LIN {X 0,Y 293.66,Z 698.302,A -85,B 0,C 180,E1 -17167.855,E2 -17167.855} C_VEL
LIN {X 0,Y 291.974,Z 709.944,A -85,B 0,C 180,E1 -17169.203,E2 -17169.203} C_VEL
LIN {X 0,Y 290.362,Z 720.316,A -85,B 0,C 180,E1 -17170.73,E2 -17170.73} C_VEL
LIN {X 0,Y 288.94,Z 728.928,A -85,B 0,C 180,E1 -17172.298,E2 -17172.298} C_VEL
LIN {X 0,Y 287.4,Z 736.795,A -85,B 0,C 180,E1 -17174.031,E2 -17174.031} C_VEL
LIN {X 0,Y 285.911,Z 744.477,A -85,B 0,C 180,E1 -17176.132,E2 -17176.132} C_VEL
LIN {X 0,Y 284.519,Z 751.531,A -85,B 0,C 180,E1 -17178.602,E2 -17178.602} C_VEL
LIN {X 0,Y 283.609,Z 756.227,A -85,B 0,C 180,E1 -17180.73,E2 -17180.73} C_VEL
LIN {X 0,Y 283.054,Z 759.814,A -85,B 0,C 180,E1 -17182.867,E2 -17182.867} C_VEL
LIN {X 0,Y 282.799,Z 761.667,A -85,B 0,C 180,E1 -17184.294,E2 -17184.294} C_VEL
LIN {X 0,Y 282.63,Z 763.061,A -85,B 0,C 180,E1 -17185.721,E2 -17185.721} C_VEL
LIN {X 0,Y 282.493,Z 764.055,A -85,B 0,C 180,E1 -17187.147,E2 -17187.147} C_VEL
LIN {X 0,Y 282.364,Z 764.898,A -85,B 0,C 180,E1 -17189.999,E2 -17189.999} C_VEL
LIN {X 0,Y 282.38,Z 764.707,A -85,B 0,C 180,E1 -17191.425,E2 -17191.425} C_VEL
LIN {X 0,Y 282.491,Z 764.121,A -85,B 0,C 180,E1 -17192.851,E2 -17192.851} C_VEL
LIN {X 0,Y 282.625,Z 763.156,A -85,B 0,C 180,E1 -17194.277,E2 -17194.277} C_VEL
LIN {X 0,Y 282.945,Z 760.817,A -85,B 0,C 180,E1 -17196.509,E2 -17196.509} C_VEL
LIN {X 0,Y 283.396,Z 757.737,A -85,B 0,C 180,E1 -17198.556,E2 -17198.556} C_VEL
LIN {X 0,Y 284.131,Z 753.485,A -85,B 0,C 180,E1 -17200.69,E2 -17200.69} C_VEL
LIN {X 0,Y 285.397,Z 747.048,A -85,B 0,C 180,E1 -17203.165,E2 -17203.165} C_VEL
LIN {X 0,Y 286.721,Z 739.97,A -85,B 0,C 180,E1 -17205.276,E2 -17205.276} C_VEL
LIN {X 0,Y 288.594,Z 731.145,A -85,B 0,C 180,E1 -17207.355,E2 -17207.355} C_VEL
LIN {X 0,Y 290.236,Z 721.447,A -85,B 0,C 180,E1 -17209.199,E2 -17209.199} C_VEL
LIN {X 0,Y 291.868,Z 710.779,A -85,B 0,C 180,E1 -17210.802,E2 -17210.802} C_VEL
LIN {X 0,Y 293.584,Z 699.328,A -85,B 0,C 180,E1 -17212.149,E2 -17212.149} C_VEL
LIN {X 0,Y 295.069,Z 687.304,A -85,B 0,C 180,E1 -17213.233,E2 -17213.233} C_VEL
LIN {X 0,Y 296.164,Z 673.903,A -85,B 0,C 180,E1 -17214.116,E2 -17214.116} C_VEL
LIN {X 0,Y 297.05,Z 661.519,A -85,B 0,C 180,E1 -17214.643,E2 -17214.643} C_VEL
LIN {X 0,Y 297.959,Z 629.003,A -85,B 0,C 180,E1 -17215.45,E2 -17215.45} C_VEL
LIN {X 0,Y 298.861,Z 588.458,A -85,B 0,C 180,E1 -17216.43,E2 -17216.43} C_VEL
LIN {X 0,Y 297.491,Z 582.733,A -85,B 0,C 180,E1 -17216.714,E2 -17216.714} C_VEL
LIN {X 0,Y 289.977,Z 564.166,A -85,B 0,C 180,E1 -17217.979,E2 -17217.979} C_VEL
LIN {X 0,Y 285.638,Z 554.659,A -85,B 0,C 180,E1 -17218.766,E2 -17218.766} C_VEL
LIN {X 0,Y 284.337,Z 549.26,A -85,B 0,C 180,E1 -17220.878,E2 -17220.878} C_VEL
LIN {X 0,Y 284.322,Z 549.07,A -85,B 0,C 180,E1 -17224.646,E2 -17224.646} C_VEL
LIN {X 0,Y 284.323,Z 549.068,A -85,B 0,C 180,E1 -17228.165,E2 -17228.165} C_VEL
LIN {X 0,Y 284.266,Z 549.077,A -85,B 0,C 180,E1 -17232.123,E2 -17232.123} C_VEL
LIN {X 0,Y 284.256,Z 549.065,A -85,B 0,C 180,E1 -17236.463,E2 -17236.463} C_VEL
LIN {X 0,Y 283.58,Z 549.163,A -85,B 0,C 180,E1 -17237.646,E2 -17237.646} C_VEL
LIN {X 0,Y 280.77,Z 549.498,A -85,B 0,C 180,E1 -17239.575,E2 -17239.575} C_VEL
LIN {X 0,Y 278.391,Z 549.786,A -85,B 0,C 180,E1 -17241.142,E2 -17241.142} C_VEL
LIN {X 0,Y 277.362,Z 549.912,A -85,B 0,C 180,E1 -17242.354,E2 -17242.354} C_VEL
LIN {X 0,Y 277.272,Z 549.925,A -85,B 0,C 180,E1 -17242.765,E2 -17242.765} C_VEL
LIN {X 0,Y 277.25,Z 549.948,A -85,B 0,C 180,E1 -17246.104,E2 -17246.104} C_VEL
LIN {X 0,Y 277.255,Z 549.95,A -85,B 0,C 180,E1 -17249.538,E2 -17249.538} C_VEL
LIN {X 0,Y 277.353,Z 549.925,A -85,B 0,C 180,E1 -17252.863,E2 -17252.863} C_VEL
LIN {X 0,Y 277.322,Z 549.936,A -85,B 0,C 180,E1 -17256.079,E2 -17256.079} C_VEL
LIN {X 0,Y 277.339,Z 549.936,A -85,B 0,C 180,E1 -17260.766,E2 -17260.766} C_VEL
LIN {X 0,Y 277.427,Z 549.919,A -85,B 0,C 180,E1 -17265.325,E2 -17265.325} C_VEL
LIN {X 0,Y 277.5,Z 549.902,A -85,B 0,C 180,E1 -17269.788,E2 -17269.788} C_VEL
LIN {X 0,Y 277.646,Z 549.898,A -85,B 0,C 180,E1 -17272.729,E2 -17272.729} C_VEL
LIN {X 0,Y 277.816,Z 549.873,A -85,B 0,C 180,E1 -17278.55,E2 -17278.55} C_VEL
LIN {X 0,Y 277.816,Z 549.876,A -85,B 0,C 180,E1 -17281.45,E2 -17281.45} C_VEL
LIN {X 0,Y 277.647,Z 549.901,A -85,B 0,C 180,E1 -17287.271,E2 -17287.271} C_VEL
LIN {X 0,Y 277.5,Z 549.902,A -85,B 0,C 180,E1 -17290.212,E2 -17290.212} C_VEL
LIN {X 0,Y 277.428,Z 549.922,A -85,B 0,C 180,E1 -17294.674,E2 -17294.674} C_VEL
LIN {X 0,Y 277.34,Z 549.939,A -85,B 0,C 180,E1 -17299.234,E2 -17299.234} C_VEL
LIN {X 0,Y 277.312,Z 549.942,A -85,B 0,C 180,E1 -17304.171,E2 -17304.171} C_VEL
LIN {X 0,Y 277.314,Z 549.934,A -85,B 0,C 180,E1 -17307.504,E2 -17307.504} C_VEL
LIN {X 0,Y 277.266,Z 549.942,A -85,B 0,C 180,E1 -17310.482,E2 -17310.482} C_VEL
LIN {X 0,Y 277.241,Z 549.947,A -85,B 0,C 180,E1 -17313.897,E2 -17313.897} C_VEL
LIN {X 0,Y 277.262,Z 549.925,A -85,B 0,C 180,E1 -17317.47,E2 -17317.47} C_VEL
LIN {X 0,Y 277.228,Z 549.942,A -85,B 0,C 180,E1 -17321.233,E2 -17321.233} C_VEL
LIN {X 0,Y 277.242,Z 549.952,A -85,B 0,C 180,E1 -17325.218,E2 -17325.218} C_VEL
LIN {X 0,Y 277.291,Z 549.942,A -85,B 0,C 180,E1 -17329.496,E2 -17329.496} C_VEL
LIN {X 0,Y 277.315,Z 549.99,A -85,B 0,C 180,E1 -17333.938,E2 -17333.938} C_VEL
LIN {X 0,Y 279.574,Z 559.685,A -85,B 0,C 180,E1 -17337.713,E2 -17337.713} C_VEL
LIN {X 0,Y 281.436,Z 568.37,A -85,B 0,C 180,E1 -17340.783,E2 -17340.783} C_VEL
LIN {X 0,Y 284.13,Z 574.997,A -85,B 0,C 180,E1 -17341.333,E2 -17341.333} C_VEL
LIN {X 0,Y 286.954,Z 582.56,A -85,B 0,C 180,E1 -17341.849,E2 -17341.849} C_VEL
LIN {X 0,Y 291.432,Z 609.842,A -85,B 0,C 180,E1 -17343.055,E2 -17343.055} C_VEL
LIN {X 0,Y 291.999,Z 615.327,A -85,B 0,C 180,E1 -17343.259,E2 -17343.259} C_VEL
LIN {X 0,Y 290.224,Z 676.927,A -85,B 0,C 180,E1 -17344.785,E2 -17344.785} C_VEL
LIN {X 0,Y 289.155,Z 690.836,A -85,B 0,C 180,E1 -17345.405,E2 -17345.405} C_VEL
LIN {X 0,Y 287.792,Z 703.287,A -85,B 0,C 180,E1 -17346.24,E2 -17346.24} C_VEL
LIN {X 0,Y 286.313,Z 714.402,A -85,B 0,C 180,E1 -17347.258,E2 -17347.258} C_VEL
LIN {X 0,Y 284.46,Z 725.973,A -85,B 0,C 180,E1 -17348.63,E2 -17348.63} C_VEL
LIN {X 0,Y 282.615,Z 736.394,A -85,B 0,C 180,E1 -17350.196,E2 -17350.196} C_VEL
LIN {X 0,Y 280.947,Z 745.535,A -85,B 0,C 180,E1 -17351.913,E2 -17351.913} C_VEL
LIN {X 0,Y 279.276,Z 754.164,A -85,B 0,C 180,E1 -17353.931,E2 -17353.931} C_VEL
LIN {X 0,Y 277.824,Z 761.597,A -85,B 0,C 180,E1 -17356.096,E2 -17356.096} C_VEL
LIN {X 0,Y 276.714,Z 767.566,A -85,B 0,C 180,E1 -17358.278,E2 -17358.278} C_VEL
LIN {X 0,Y 275.962,Z 772.287,A -85,B 0,C 180,E1 -17360.473,E2 -17360.473} C_VEL
LIN {X 0,Y 275.495,Z 775.9,A -85,B 0,C 180,E1 -17362.673,E2 -17362.673} C_VEL
LIN {X 0,Y 275.263,Z 778.342,A -85,B 0,C 180,E1 -17364.715,E2 -17364.715} C_VEL
LIN {X 0,Y 275.255,Z 780.158,A -85,B 0,C 180,E1 -17367.074,E2 -17367.074} C_VEL
LIN {X 0,Y 275.249,Z 781.14,A -85,B 0,C 180,E1 -17370.001,E2 -17370.001} C_VEL
LIN {X 0,Y 275.241,Z 782.664,A -85,B 0,C 180,E1 -17371.464,E2 -17371.464} C_VEL
LIN {X 0,Y 275.272,Z 783.614,A -85,B 0,C 180,E1 -17372.928,E2 -17372.928} C_VEL
LIN {X 0,Y 275.324,Z 783.939,A -85,B 0,C 180,E1 -17374.393,E2 -17374.393} C_VEL
LIN {X 0,Y 275.495,Z 783.663,A -85,B 0,C 180,E1 -17375.858,E2 -17375.858} C_VEL
LIN {X 0,Y 275.784,Z 782.827,A -85,B 0,C 180,E1 -17377.322,E2 -17377.322} C_VEL
LIN {X 0,Y 276.479,Z 780.557,A -85,B 0,C 180,E1 -17379.512,E2 -17379.512} C_VEL
LIN {X 0,Y 277.48,Z 776.829,A -85,B 0,C 180,E1 -17381.692,E2 -17381.692} C_VEL
LIN {X 0,Y 278.737,Z 771.632,A -85,B 0,C 180,E1 -17383.86,E2 -17383.86} C_VEL
LIN {X 0,Y 280.153,Z 765.979,A -85,B 0,C 180,E1 -17385.646,E2 -17385.646} C_VEL
LIN {X 0,Y 281.707,Z 758.788,A -85,B 0,C 180,E1 -17387.421,E2 -17387.421} C_VEL
LIN {X 0,Y 283.291,Z 750.413,A -85,B 0,C 180,E1 -17389.084,E2 -17389.084} C_VEL
LIN {X 0,Y 284.767,Z 740.738,A -85,B 0,C 180,E1 -17390.592,E2 -17390.592} C_VEL
LIN {X 0,Y 286.137,Z 730.818,A -85,B 0,C 180,E1 -17391.809,E2 -17391.809} C_VEL
LIN {X 0,Y 287.279,Z 719.702,A -85,B 0,C 180,E1 -17392.854,E2 -17392.854} C_VEL
LIN {X 0,Y 288.01,Z 708.239,A -85,B 0,C 180,E1 -17393.649,E2 -17393.649} C_VEL
LIN {X 0,Y 289.321,Z 688.909,A -85,B 0,C 180,E1 -17394.679,E2 -17394.679} C_VEL
LIN {X 0,Y 292.046,Z 660.371,A -85,B 0,C 180,E1 -17396.005,E2 -17396.005} C_VEL
LIN {X 0,Y 295.2,Z 631.603,A -85,B 0,C 180,E1 -17397.326,E2 -17397.326} C_VEL
LIN {X 0,Y 299.314,Z 618.162,A -85,B 0,C 180,E1 -17398.552,E2 -17398.552} C_VEL
LIN {X 0,Y 302.154,Z 605.802,A -85,B 0,C 180,E1 -17400.159,E2 -17400.159} C_VEL
LIN {X 0,Y 302.686,Z 602.213,A -85,B 0,C 180,E1 -17400.785,E2 -17400.785} C_VEL
LIN {X 0,Y 302.288,Z 595.852,A -85,B 0,C 180,E1 -17402.573,E2 -17402.573} C_VEL
LIN {X 0,Y 302.131,Z 592.975,A -85,B 0,C 180,E1 -17403.513,E2 -17403.513} C_VEL
LIN {X 0,Y 301.865,Z 592.038,A -85,B 0,C 180,E1 -17403.972,E2 -17403.972} C_VEL
LIN {X 0,Y 300.413,Z 589.492,A -85,B 0,C 180,E1 -17405.794,E2 -17405.794} C_VEL
LIN {X 0,Y 299.249,Z 587.817,A -85,B 0,C 180,E1 -17407.636,E2 -17407.636} C_VEL
LIN {X 0,Y 297.898,Z 586.526,A -85,B 0,C 180,E1 -17410.979,E2 -17410.979} C_VEL
LIN {X 0,Y 297.615,Z 586.677,A -85,B 0,C 180,E1 -17413.223,E2 -17413.223} C_VEL
LIN {X 0,Y 297.632,Z 587.564,A -85,B 0,C 180,E1 -17415.105,E2 -17415.105} C_VEL
LIN {X 0,Y 297.839,Z 589.148,A -85,B 0,C 180,E1 -17417.013,E2 -17417.013} C_VEL
LIN {X 0,Y 298.519,Z 592.562,A -85,B 0,C 180,E1 -17419.79,E2 -17419.79} C_VEL
LIN {X 0,Y 299.2,Z 597.104,A -85,B 0,C 180,E1 -17422.358,E2 -17422.358} C_VEL
LIN {X 0,Y 299.735,Z 602.203,A -85,B 0,C 180,E1 -17424.609,E2 -17424.609} C_VEL
LIN {X 0,Y 299.975,Z 606.139,A -85,B 0,C 180,E1 -17426.091,E2 -17426.091} C_VEL
LIN {X 0,Y 299.541,Z 608.357,A -85,B 0,C 180,E1 -17426.691,E2 -17426.691} C_VEL
LIN {X 0,Y 294.292,Z 628.859,A -85,B 0,C 180,E1 -17431.47,E2 -17431.47} C_VEL
LIN {X 0,Y 293.568,Z 632.929,A -85,B 0,C 180,E1 -17432.349,E2 -17432.349} C_VEL
LIN {X 0,Y 296.081,Z 648.237,A -85,B 0,C 180,E1 -17434.027,E2 -17434.027} C_VEL
LIN {X 0,Y 297.588,Z 660.605,A -85,B 0,C 180,E1 -17435.133,E2 -17435.133} C_VEL
LIN {X 0,Y 297.812,Z 664.77,A -85,B 0,C 180,E1 -17435.442,E2 -17435.442} C_VEL
LIN {X 0,Y 293.678,Z 707.804,A -85,B 0,C 180,E1 -17437.301,E2 -17437.301} C_VEL
LIN {X 0,Y 292.176,Z 719.062,A -85,B 0,C 180,E1 -17438.016,E2 -17438.016} C_VEL
LIN {X 0,Y 290.176,Z 730.518,A -85,B 0,C 180,E1 -17439.069,E2 -17439.069} C_VEL
LIN {X 0,Y 288.204,Z 740.099,A -85,B 0,C 180,E1 -17440.224,E2 -17440.224} C_VEL
LIN {X 0,Y 286.358,Z 747.778,A -85,B 0,C 180,E1 -17441.394,E2 -17441.394} C_VEL
LIN {X 0,Y 284.507,Z 754.948,A -85,B 0,C 180,E1 -17442.757,E2 -17442.757} C_VEL
LIN {X 0,Y 282.39,Z 762.252,A -85,B 0,C 180,E1 -17444.482,E2 -17444.482} C_VEL
LIN {X 0,Y 280.492,Z 767.926,A -85,B 0,C 180,E1 -17446.23,E2 -17446.23} C_VEL
LIN {X 0,Y 278.74,Z 773.106,A -85,B 0,C 180,E1 -17448.363,E2 -17448.363} C_VEL
LIN {X 0,Y 277.815,Z 775.691,A -85,B 0,C 180,E1 -17449.8,E2 -17449.8} C_VEL
LIN {X 0,Y 276.639,Z 778.686,A -85,B 0,C 180,E1 -17452.225,E2 -17452.225} C_VEL
LIN {X 0,Y 275.964,Z 779.813,A -85,B 0,C 180,E1 -17454.153,E2 -17454.153} C_VEL
LIN {X 0,Y 275.56,Z 780.051,A -85,B 0,C 180,E1 -17455.612,E2 -17455.612} C_VEL
LIN {X 0,Y 275.358,Z 779.681,A -85,B 0,C 180,E1 -17457.074,E2 -17457.074} C_VEL
LIN {X 0,Y 275.252,Z 778.702,A -85,B 0,C 180,E1 -17458.537,E2 -17458.537} C_VEL
LIN {X 0,Y 275.21,Z 776.131,A -85,B 0,C 180,E1 -17460.732,E2 -17460.732} C_VEL
LIN {X 0,Y 275.385,Z 772.08,A -85,B 0,C 180,E1 -17462.926,E2 -17462.926} C_VEL
LIN {X 0,Y 275.5,Z 767.367,A -85,B 0,C 180,E1 -17464.802,E2 -17464.802} C_VEL
LIN {X 0,Y 275.72,Z 761.729,A -85,B 0,C 180,E1 -17466.513,E2 -17466.513} C_VEL
LIN {X 0,Y 276.092,Z 755.384,A -85,B 0,C 180,E1 -17468.048,E2 -17468.048} C_VEL
LIN {X 0,Y 276.46,Z 747.97,A -85,B 0,C 180,E1 -17469.511,E2 -17469.511} C_VEL
LIN {X 0,Y 276.958,Z 738.718,A -85,B 0,C 180,E1 -17470.971,E2 -17470.971} C_VEL
LIN {X 0,Y 277.463,Z 729.843,A -85,B 0,C 180,E1 -17472.062,E2 -17472.062} C_VEL
LIN {X 0,Y 277.951,Z 719.501,A -85,B 0,C 180,E1 -17473.061,E2 -17473.061} C_VEL
LIN {X 0,Y 278.328,Z 708.075,A -85,B 0,C 180,E1 -17473.833,E2 -17473.833} C_VEL
LIN {X 0,Y 278.666,Z 694.962,A -85,B 0,C 180,E1 -17474.421,E2 -17474.421} C_VEL
LIN {X 0,Y 279.588,Z 654.121,A -85,B 0,C 180,E1 -17476.029,E2 -17476.029} C_VEL
LIN {X 0,Y 278.107,Z 632.469,A -85,B 0,C 180,E1 -17476.921,E2 -17476.921} C_VEL
LIN {X 0,Y 278.379,Z 628.581,A -85,B 0,C 180,E1 -17477.635,E2 -17477.635} C_VEL
LIN {X 0,Y 279.838,Z 608.07,A -85,B 0,C 180,E1 -17481.876,E2 -17481.876} C_VEL
LIN {X 0,Y 281.515,Z 586.927,A -85,B 0,C 180,E1 -17486.242,E2 -17486.242} C_VEL
LIN {X 0,Y 282.506,Z 575.81,A -85,B 0,C 180,E1 -17488.536,E2 -17488.536} C_VEL
LIN {X 0,Y 281.422,Z 569.277,A -85,B 0,C 180,E1 -17489.965,E2 -17489.965} C_VEL
LIN {X 0,Y 277.347,Z 550.123,A -85,B 0,C 180,E1 -17494.348,E2 -17494.348} C_VEL
LIN {X 0,Y 277.276,Z 549.948,A -85,B 0,C 180,E1 -17498.209,E2 -17498.209} C_VEL
LIN {X 0,Y 277.222,Z 549.902,A -85,B 0,C 180,E1 -17502.675,E2 -17502.675} C_VEL
LIN {X 0,Y 277.24,Z 549.953,A -85,B 0,C 180,E1 -17506.807,E2 -17506.807} C_VEL
LIN {X 0,Y 277.239,Z 549.916,A -85,B 0,C 180,E1 -17510.671,E2 -17510.671} C_VEL
LIN {X 0,Y 277.288,Z 549.938,A -85,B 0,C 180,E1 -17514.341,E2 -17514.341} C_VEL
LIN {X 0,Y 277.316,Z 550.144,A -85,B 0,C 180,E1 -17518.646,E2 -17518.646} C_VEL
LIN {X 0,Y 278.458,Z 554.86,A -85,B 0,C 180,E1 -17520.544,E2 -17520.544} C_VEL
LIN {X 0,Y 282.633,Z 563.933,A -85,B 0,C 180,E1 -17521.338,E2 -17521.338} C_VEL
LIN {X 0,Y 289.849,Z 581.09,A -85,B 0,C 180,E1 -17522.593,E2 -17522.593} C_VEL
LIN {X 0,Y 292.051,Z 587.521,A -85,B 0,C 180,E1 -17522.993,E2 -17522.993} C_VEL
LIN {X 0,Y 292.601,Z 590.728,A -85,B 0,C 180,E1 -17523.136,E2 -17523.136} C_VEL
LIN {X 0,Y 290.489,Z 661.08,A -85,B 0,C 180,E1 -17524.854,E2 -17524.854} C_VEL
LIN {X 0,Y 289.618,Z 674.452,A -85,B 0,C 180,E1 -17525.444,E2 -17525.444} C_VEL
LIN {X 0,Y 288.495,Z 687.2,A -85,B 0,C 180,E1 -17526.298,E2 -17526.298} C_VEL
LIN {X 0,Y 287.105,Z 698.512,A -85,B 0,C 180,E1 -17527.321,E2 -17527.321} C_VEL
LIN {X 0,Y 285.349,Z 710.153,A -85,B 0,C 180,E1 -17528.697,E2 -17528.697} C_VEL
LIN {X 0,Y 283.569,Z 721.131,A -85,B 0,C 180,E1 -17530.356,E2 -17530.356} C_VEL
LIN {X 0,Y 281.854,Z 730.827,A -85,B 0,C 180,E1 -17532.213,E2 -17532.213} C_VEL
LIN {X 0,Y 279.978,Z 739.737,A -85,B 0,C 180,E1 -17534.344,E2 -17534.344} C_VEL
LIN {X 0,Y 278.551,Z 746.904,A -85,B 0,C 180,E1 -17536.502,E2 -17536.502} C_VEL
LIN {X 0,Y 277.542,Z 751.738,A -85,B 0,C 180,E1 -17538.311,E2 -17538.311} C_VEL
LIN {X 0,Y 276.585,Z 756.434,A -85,B 0,C 180,E1 -17540.492,E2 -17540.492} C_VEL
LIN {X 0,Y 276.009,Z 760.02,A -85,B 0,C 180,E1 -17542.684,E2 -17542.684} C_VEL
LIN {X 0,Y 275.724,Z 761.873,A -85,B 0,C 180,E1 -17544.147,E2 -17544.147} C_VEL
LIN {X 0,Y 275.557,Z 763.266,A -85,B 0,C 180,E1 -17545.61,E2 -17545.61} C_VEL
LIN {X 0,Y 275.427,Z 764.259,A -85,B 0,C 180,E1 -17547.073,E2 -17547.073} C_VEL
LIN {X 0,Y 275.286,Z 765.102,A -85,B 0,C 180,E1 -17549.999,E2 -17549.999} C_VEL
LIN {X 0,Y 275.306,Z 764.911,A -85,B 0,C 180,E1 -17551.461,E2 -17551.461} C_VEL
LIN {X 0,Y 275.424,Z 764.325,A -85,B 0,C 180,E1 -17552.924,E2 -17552.924} C_VEL
LIN {X 0,Y 275.552,Z 763.36,A -85,B 0,C 180,E1 -17554.387,E2 -17554.387} C_VEL
LIN {X 0,Y 275.861,Z 761.246,A -85,B 0,C 180,E1 -17556.49,E2 -17556.49} C_VEL
LIN {X 0,Y 276.386,Z 757.941,A -85,B 0,C 180,E1 -17558.774,E2 -17558.774} C_VEL
LIN {X 0,Y 277.15,Z 753.689,A -85,B 0,C 180,E1 -17560.962,E2 -17560.962} C_VEL
LIN {X 0,Y 278.495,Z 747.25,A -85,B 0,C 180,E1 -17563.498,E2 -17563.498} C_VEL
LIN {X 0,Y 279.884,Z 740.172,A -85,B 0,C 180,E1 -17565.659,E2 -17565.659} C_VEL
LIN {X 0,Y 281.84,Z 731.346,A -85,B 0,C 180,E1 -17567.785,E2 -17567.785} C_VEL
LIN {X 0,Y 283.546,Z 721.622,A -85,B 0,C 180,E1 -17569.675,E2 -17569.675} C_VEL
LIN {X 0,Y 285.249,Z 710.979,A -85,B 0,C 180,E1 -17571.308,E2 -17571.308} C_VEL
LIN {X 0,Y 287.026,Z 699.527,A -85,B 0,C 180,E1 -17572.682,E2 -17572.682} C_VEL
LIN {X 0,Y 288.578,Z 687.5,A -85,B 0,C 180,E1 -17573.787,E2 -17573.787} C_VEL
LIN {X 0,Y 289.721,Z 674.097,A -85,B 0,C 180,E1 -17574.687,E2 -17574.687} C_VEL
LIN {X 0,Y 290.622,Z 661.708,A -85,B 0,C 180,E1 -17575.226,E2 -17575.226} C_VEL
LIN {X 0,Y 291.657,Z 625.335,A -85,B 0,C 180,E1 -17576.144,E2 -17576.144} C_VEL
LIN {X 0,Y 292.558,Z 589.851,A -85,B 0,C 180,E1 -17577.012,E2 -17577.012} C_VEL
LIN {X 0,Y 291.498,Z 585.387,A -85,B 0,C 180,E1 -17577.241,E2 -17577.241} C_VEL
LIN {X 0,Y 284.212,Z 567.439,A -85,B 0,C 180,E1 -17578.51,E2 -17578.51} C_VEL
LIN {X 0,Y 278.49,Z 554.972,A -85,B 0,C 180,E1 -17579.565,E2 -17579.565} C_VEL
LIN {X 0,Y 277.736,Z 552.086,A -85,B 0,C 180,E1 -17580.643,E2 -17580.643} C_VEL
LIN {X 0,Y 277.276,Z 549.963,A -85,B 0,C 180,E1 -17581.676,E2 -17581.676} C_VEL
LIN {X 0,Y 277.323,Z 549.932,A -85,B 0,C 180,E1 -17585.81,E2 -17585.81} C_VEL
LIN {X 0,Y 277.236,Z 549.939,A -85,B 0,C 180,E1 -17589.326,E2 -17589.326} C_VEL
LIN {X 0,Y 277.205,Z 549.949,A -85,B 0,C 180,E1 -17593.197,E2 -17593.197} C_VEL
LIN {X 0,Y 277.232,Z 549.95,A -85,B 0,C 180,E1 -17597.319,E2 -17597.319} C_VEL
LIN {X 0,Y 277.261,Z 549.922,A -85,B 0,C 180,E1 -17600.676,E2 -17600.676} C_VEL
LIN {X 0,Y 277.272,Z 549.925,A -85,B 0,C 180,E1 -17602.765,E2 -17602.765} C_VEL
LIN {X 0,Y 276.591,Z 550.026,A -85,B 0,C 180,E1 -17603.978,E2 -17603.978} C_VEL
LIN {X 0,Y 273.74,Z 550.386,A -85,B 0,C 180,E1 -17605.954,E2 -17605.954} C_VEL
LIN {X 0,Y 271.324,Z 550.689,A -85,B 0,C 180,E1 -17607.559,E2 -17607.559} C_VEL
LIN {X 0,Y 270.281,Z 550.817,A -85,B 0,C 180,E1 -17608.803,E2 -17608.803} C_VEL
LIN {X 0,Y 270.192,Z 550.826,A -85,B 0,C 180,E1 -17609.225,E2 -17609.225} C_VEL
LIN {X 0,Y 270.259,Z 550.808,A -85,B 0,C 180,E1 -17612.145,E2 -17612.145} C_VEL
LIN {X 0,Y 270.271,Z 550.818,A -85,B 0,C 180,E1 -17615.518,E2 -17615.518} C_VEL
LIN {X 0,Y 270.295,Z 550.814,A -85,B 0,C 180,E1 -17620.244,E2 -17620.244} C_VEL
LIN {X 0,Y 270.396,Z 550.792,A -85,B 0,C 180,E1 -17624.935,E2 -17624.935} C_VEL
LIN {X 0,Y 270.435,Z 550.783,A -85,B 0,C 180,E1 -17629.519,E2 -17629.519} C_VEL
LIN {X 0,Y 270.604,Z 550.775,A -85,B 0,C 180,E1 -17632.539,E2 -17632.539} C_VEL
LIN {X 0,Y 270.781,Z 550.749,A -85,B 0,C 180,E1 -17638.513,E2 -17638.513} C_VEL
LIN {X 0,Y 270.781,Z 550.752,A -85,B 0,C 180,E1 -17641.487,E2 -17641.487} C_VEL
LIN {X 0,Y 270.605,Z 550.778,A -85,B 0,C 180,E1 -17647.461,E2 -17647.461} C_VEL
LIN {X 0,Y 270.435,Z 550.783,A -85,B 0,C 180,E1 -17650.481,E2 -17650.481} C_VEL
LIN {X 0,Y 270.396,Z 550.795,A -85,B 0,C 180,E1 -17655.065,E2 -17655.065} C_VEL
LIN {X 0,Y 270.296,Z 550.814,A -85,B 0,C 180,E1 -17659.756,E2 -17659.756} C_VEL
LIN {X 0,Y 270.267,Z 550.819,A -85,B 0,C 180,E1 -17664.586,E2 -17664.586} C_VEL
LIN {X 0,Y 270.262,Z 550.817,A -85,B 0,C 180,E1 -17667.91,E2 -17667.91} C_VEL
LIN {X 0,Y 270.178,Z 550.823,A -85,B 0,C 180,E1 -17671.349,E2 -17671.349} C_VEL
LIN {X 0,Y 270.196,Z 550.814,A -85,B 0,C 180,E1 -17674.906,E2 -17674.906} C_VEL
LIN {X 0,Y 270.217,Z 550.821,A -85,B 0,C 180,E1 -17678.718,E2 -17678.718} C_VEL
LIN {X 0,Y 270.19,Z 550.81,A -85,B 0,C 180,E1 -17682.555,E2 -17682.555} C_VEL
LIN {X 0,Y 270.209,Z 550.814,A -85,B 0,C 180,E1 -17686.741,E2 -17686.741} C_VEL
LIN {X 0,Y 270.245,Z 550.82,A -85,B 0,C 180,E1 -17689.449,E2 -17689.449} C_VEL
LIN {X 0,Y 270.252,Z 550.877,A -85,B 0,C 180,E1 -17693.266,E2 -17693.266} C_VEL
LIN {X 0,Y 272.164,Z 558.933,A -85,B 0,C 180,E1 -17696.538,E2 -17696.538} C_VEL
LIN {X 0,Y 274.21,Z 568.209,A -85,B 0,C 180,E1 -17699.945,E2 -17699.945} C_VEL
LIN {X 0,Y 278.369,Z 578.133,A -85,B 0,C 180,E1 -17700.778,E2 -17700.778} C_VEL
LIN {X 0,Y 280.93,Z 584.879,A -85,B 0,C 180,E1 -17701.26,E2 -17701.26} C_VEL
LIN {X 0,Y 285.405,Z 612.982,A -85,B 0,C 180,E1 -17702.531,E2 -17702.531} C_VEL
LIN {X 0,Y 285.61,Z 617.978,A -85,B 0,C 180,E1 -17702.69,E2 -17702.69} C_VEL
LIN {X 0,Y 283.814,Z 676.736,A -85,B 0,C 180,E1 -17704.174,E2 -17704.174} C_VEL
LIN {X 0,Y 282.728,Z 690.64,A -85,B 0,C 180,E1 -17704.807,E2 -17704.807} C_VEL
LIN {X 0,Y 281.308,Z 703.089,A -85,B 0,C 180,E1 -17705.657,E2 -17705.657} C_VEL
LIN {X 0,Y 279.521,Z 715.787,A -85,B 0,C 180,E1 -17706.869,E2 -17706.869} C_VEL
LIN {X 0,Y 277.652,Z 727.067,A -85,B 0,C 180,E1 -17708.274,E2 -17708.274} C_VEL
LIN {X 0,Y 275.727,Z 737.23,A -85,B 0,C 180,E1 -17709.875,E2 -17709.875} C_VEL
LIN {X 0,Y 274.052,Z 745.989,A -85,B 0,C 180,E1 -17711.597,E2 -17711.597} C_VEL
LIN {X 0,Y 272.428,Z 753.961,A -85,B 0,C 180,E1 -17713.516,E2 -17713.516} C_VEL
LIN {X 0,Y 270.913,Z 761.393,A -85,B 0,C 180,E1 -17715.734,E2 -17715.734} C_VEL
LIN {X 0,Y 269.714,Z 767.361,A -85,B 0,C 180,E1 -17717.969,E2 -17717.969} C_VEL
LIN {X 0,Y 268.946,Z 772.083,A -85,B 0,C 180,E1 -17720.222,E2 -17720.222} C_VEL
LIN {X 0,Y 268.42,Z 775.695,A -85,B 0,C 180,E1 -17722.479,E2 -17722.479} C_VEL
LIN {X 0,Y 268.178,Z 778.333,A -85,B 0,C 180,E1 -17724.777,E2 -17724.777} C_VEL
LIN {X 0,Y 268.167,Z 779.953,A -85,B 0,C 180,E1 -17726.997,E2 -17726.997} C_VEL
LIN {X 0,Y 268.181,Z 780.561,A -85,B 0,C 180,E1 -17728.5,E2 -17728.5} C_VEL
LIN {X 0,Y 268.156,Z 781.04,A -85,B 0,C 180,E1 -17730.377,E2 -17730.377} C_VEL
LIN {X 0,Y 268.169,Z 782.254,A -85,B 0,C 180,E1 -17731.503,E2 -17731.503} C_VEL
LIN {X 0,Y 268.187,Z 783.31,A -85,B 0,C 180,E1 -17733.006,E2 -17733.006} C_VEL
LIN {X 0,Y 268.355,Z 783.792,A -85,B 0,C 180,E1 -17735.621,E2 -17735.621} C_VEL
LIN {X 0,Y 268.738,Z 783.047,A -85,B 0,C 180,E1 -17737.515,E2 -17737.515} C_VEL
LIN {X 0,Y 269.194,Z 781.851,A -85,B 0,C 180,E1 -17739.014,E2 -17739.014} C_VEL
LIN {X 0,Y 270.194,Z 778.888,A -85,B 0,C 180,E1 -17741.251,E2 -17741.251} C_VEL
LIN {X 0,Y 271.509,Z 774.576,A -85,B 0,C 180,E1 -17743.473,E2 -17743.473} C_VEL
LIN {X 0,Y 272.824,Z 769.751,A -85,B 0,C 180,E1 -17745.311,E2 -17745.311} C_VEL
LIN {X 0,Y 274.474,Z 763.582,A -85,B 0,C 180,E1 -17747.126,E2 -17747.126} C_VEL
LIN {X 0,Y 276.272,Z 755.922,A -85,B 0,C 180,E1 -17748.927,E2 -17748.927} C_VEL
LIN {X 0,Y 277.962,Z 747.422,A -85,B 0,C 180,E1 -17750.522,E2 -17750.522} C_VEL
LIN {X 0,Y 279.439,Z 739.295,A -85,B 0,C 180,E1 -17751.738,E2 -17751.738} C_VEL
LIN {X 0,Y 280.766,Z 730.378,A -85,B 0,C 180,E1 -17752.831,E2 -17752.831} C_VEL
LIN {X 0,Y 282.07,Z 719.288,A -85,B 0,C 180,E1 -17753.885,E2 -17753.885} C_VEL
LIN {X 0,Y 282.995,Z 707.47,A -85,B 0,C 180,E1 -17754.729,E2 -17754.729} C_VEL
LIN {X 0,Y 284.631,Z 686.199,A -85,B 0,C 180,E1 -17755.848,E2 -17755.848} C_VEL
LIN {X 0,Y 287.617,Z 659.501,A -85,B 0,C 180,E1 -17757.122,E2 -17757.122} C_VEL
LIN {X 0,Y 290.778,Z 632.039,A -85,B 0,C 180,E1 -17758.415,E2 -17758.415} C_VEL
LIN {X 0,Y 294.937,Z 619.147,A -85,B 0,C 180,E1 -17759.635,E2 -17759.635} C_VEL
LIN {X 0,Y 297.935,Z 607.271,A -85,B 0,C 180,E1 -17761.264,E2 -17761.264} C_VEL
LIN {X 0,Y 297.992,Z 604.716,A -85,B 0,C 180,E1 -17761.892,E2 -17761.892} C_VEL
LIN {X 0,Y 297.791,Z 599.086,A -85,B 0,C 180,E1 -17763.605,E2 -17763.605} C_VEL
LIN {X 0,Y 297.576,Z 597.535,A -85,B 0,C 180,E1 -17764.248,E2 -17764.248} C_VEL
LIN {X 0,Y 295.937,Z 594.701,A -85,B 0,C 180,E1 -17766.422,E2 -17766.422} C_VEL
LIN {X 0,Y 294.746,Z 593.212,A -85,B 0,C 180,E1 -17768.314,E2 -17768.314} C_VEL
LIN {X 0,Y 293.928,Z 592.438,A -85,B 0,C 180,E1 -17770.211,E2 -17770.211} C_VEL
LIN {X 0,Y 293.442,Z 592.216,A -85,B 0,C 180,E1 -17772.115,E2 -17772.115} C_VEL
LIN {X 0,Y 293.267,Z 592.671,A -85,B 0,C 180,E1 -17774.033,E2 -17774.033} C_VEL
LIN {X 0,Y 293.249,Z 593.836,A -85,B 0,C 180,E1 -17775.972,E2 -17775.972} C_VEL
LIN {X 0,Y 293.672,Z 596.972,A -85,B 0,C 180,E1 -17778.985,E2 -17778.985} C_VEL
LIN {X 0,Y 294.203,Z 601.07,A -85,B 0,C 180,E1 -17781.604,E2 -17781.604} C_VEL
LIN {X 0,Y 294.514,Z 604.676,A -85,B 0,C 180,E1 -17783.375,E2 -17783.375} C_VEL
LIN {X 0,Y 294.711,Z 610.018,A -85,B 0,C 180,E1 -17785.545,E2 -17785.545} C_VEL
LIN {X 0,Y 293.993,Z 612.772,A -85,B 0,C 180,E1 -17786.276,E2 -17786.276} C_VEL
LIN {X 0,Y 288.622,Z 632.618,A -85,B 0,C 180,E1 -17790.997,E2 -17790.997} C_VEL
LIN {X 0,Y 290.892,Z 647.171,A -85,B 0,C 180,E1 -17792.734,E2 -17792.734} C_VEL
LIN {X 0,Y 292.363,Z 659.834,A -85,B 0,C 180,E1 -17793.99,E2 -17793.99} C_VEL
LIN {X 0,Y 292.78,Z 666.126,A -85,B 0,C 180,E1 -17794.499,E2 -17794.499} C_VEL
LIN {X 0,Y 288.435,Z 707.668,A -85,B 0,C 180,E1 -17796.342,E2 -17796.342} C_VEL
LIN {X 0,Y 286.745,Z 719.32,A -85,B 0,C 180,E1 -17797.102,E2 -17797.102} C_VEL
LIN {X 0,Y 284.803,Z 729.939,A -85,B 0,C 180,E1 -17798.085,E2 -17798.085} C_VEL
LIN {X 0,Y 282.685,Z 739.679,A -85,B 0,C 180,E1 -17799.251,E2 -17799.251} C_VEL
LIN {X 0,Y 280.395,Z 748.365,A -85,B 0,C 180,E1 -17800.603,E2 -17800.603} C_VEL
LIN {X 0,Y 278.398,Z 755.386,A -85,B 0,C 180,E1 -17801.986,E2 -17801.986} C_VEL
LIN {X 0,Y 276.133,Z 762.603,A -85,B 0,C 180,E1 -17803.742,E2 -17803.742} C_VEL
LIN {X 0,Y 274.507,Z 767.235,A -85,B 0,C 180,E1 -17805.166,E2 -17805.166} C_VEL
LIN {X 0,Y 273.038,Z 771.034,A -85,B 0,C 180,E1 -17806.605,E2 -17806.605} C_VEL
LIN {X 0,Y 271.381,Z 775.276,A -85,B 0,C 180,E1 -17808.8,E2 -17808.8} C_VEL
LIN {X 0,Y 270.023,Z 778.19,A -85,B 0,C 180,E1 -17811.016,E2 -17811.016} C_VEL
LIN {X 0,Y 269.438,Z 779.361,A -85,B 0,C 180,E1 -17812.506,E2 -17812.506} C_VEL
LIN {X 0,Y 268.907,Z 779.973,A -85,B 0,C 180,E1 -17813.999,E2 -17813.999} C_VEL
LIN {X 0,Y 268.482,Z 780.026,A -85,B 0,C 180,E1 -17815.496,E2 -17815.496} C_VEL
LIN {X 0,Y 268.277,Z 779.52,A -85,B 0,C 180,E1 -17816.997,E2 -17816.997} C_VEL
LIN {X 0,Y 268.182,Z 778.437,A -85,B 0,C 180,E1 -17818.498,E2 -17818.498} C_VEL
LIN {X 0,Y 268.138,Z 775.561,A -85,B 0,C 180,E1 -17820.751,E2 -17820.751} C_VEL
LIN {X 0,Y 268.326,Z 771.3,A -85,B 0,C 180,E1 -17823.003,E2 -17823.003} C_VEL
LIN {X 0,Y 268.452,Z 766.485,A -85,B 0,C 180,E1 -17824.852,E2 -17824.852} C_VEL
LIN {X 0,Y 268.721,Z 760.015,A -85,B 0,C 180,E1 -17826.759,E2 -17826.759} C_VEL
LIN {X 0,Y 269.099,Z 753.724,A -85,B 0,C 180,E1 -17828.259,E2 -17828.259} C_VEL
LIN {X 0,Y 269.566,Z 744.872,A -85,B 0,C 180,E1 -17829.946,E2 -17829.946} C_VEL
LIN {X 0,Y 270.006,Z 736.07,A -85,B 0,C 180,E1 -17831.258,E2 -17831.258} C_VEL
LIN {X 0,Y 270.532,Z 726.654,A -85,B 0,C 180,E1 -17832.376,E2 -17832.376} C_VEL
LIN {X 0,Y 270.911,Z 716.022,A -85,B 0,C 180,E1 -17833.311,E2 -17833.311} C_VEL
LIN {X 0,Y 271.418,Z 704.29,A -85,B 0,C 180,E1 -17834.049,E2 -17834.049} C_VEL
LIN {X 0,Y 272.506,Z 654.424,A -85,B 0,C 180,E1 -17836.096,E2 -17836.096} C_VEL
LIN {X 0,Y 271.038,Z 632.608,A -85,B 0,C 180,E1 -17837.028,E2 -17837.028} C_VEL
LIN {X 0,Y 271.146,Z 630.622,A -85,B 0,C 180,E1 -17837.341,E2 -17837.341} C_VEL
LIN {X 0,Y 272.619,Z 610.644,A -85,B 0,C 180,E1 -17841.555,E2 -17841.555} C_VEL
LIN {X 0,Y 274.395,Z 588.696,A -85,B 0,C 180,E1 -17846.169,E2 -17846.169} C_VEL
LIN {X 0,Y 275.446,Z 577.2,A -85,B 0,C 180,E1 -17848.582,E2 -17848.582} C_VEL
LIN {X 0,Y 275.051,Z 573.585,A -85,B 0,C 180,E1 -17849.378,E2 -17849.378} C_VEL
LIN {X 0,Y 271.771,Z 558.173,A -85,B 0,C 180,E1 -17852.892,E2 -17852.892} C_VEL
LIN {X 0,Y 270.288,Z 550.989,A -85,B 0,C 180,E1 -17854.613,E2 -17854.613} C_VEL
LIN {X 0,Y 270.202,Z 550.826,A -85,B 0,C 180,E1 -17858.71,E2 -17858.71} C_VEL
LIN {X 0,Y 270.176,Z 550.779,A -85,B 0,C 180,E1 -17863.25,E2 -17863.25} C_VEL
LIN {X 0,Y 270.199,Z 550.827,A -85,B 0,C 180,E1 -17867.446,E2 -17867.446} C_VEL
LIN {X 0,Y 270.211,Z 550.795,A -85,B 0,C 180,E1 -17871.374,E2 -17871.374} C_VEL
LIN {X 0,Y 270.206,Z 550.814,A -85,B 0,C 180,E1 -17875.094,E2 -17875.094} C_VEL
LIN {X 0,Y 270.259,Z 551.04,A -85,B 0,C 180,E1 -17878.004,E2 -17878.004} C_VEL
LIN {X 0,Y 271.227,Z 555.055,A -85,B 0,C 180,E1 -17879.669,E2 -17879.669} C_VEL
LIN {X 0,Y 275.224,Z 563.584,A -85,B 0,C 180,E1 -17880.473,E2 -17880.473} C_VEL
LIN {X 0,Y 281.948,Z 578.843,A -85,B 0,C 180,E1 -17881.685,E2 -17881.685} C_VEL
LIN {X 0,Y 286.029,Z 590.075,A -85,B 0,C 180,E1 -17882.442,E2 -17882.442} C_VEL
LIN {X 0,Y 286.166,Z 594.456,A -85,B 0,C 180,E1 -17882.578,E2 -17882.578} C_VEL
LIN {X 0,Y 284.099,Z 661.301,A -85,B 0,C 180,E1 -17884.248,E2 -17884.248} C_VEL
LIN {X 0,Y 283.204,Z 674.666,A -85,B 0,C 180,E1 -17884.85,E2 -17884.85} C_VEL
LIN {X 0,Y 282.015,Z 687.412,A -85,B 0,C 180,E1 -17885.719,E2 -17885.719} C_VEL
LIN {X 0,Y 280.586,Z 698.721,A -85,B 0,C 180,E1 -17886.764,E2 -17886.764} C_VEL
LIN {X 0,Y 278.753,Z 710.362,A -85,B 0,C 180,E1 -17888.167,E2 -17888.167} C_VEL
LIN {X 0,Y 276.957,Z 720.897,A -85,B 0,C 180,E1 -17889.787,E2 -17889.787} C_VEL
LIN {X 0,Y 275.467,Z 729.343,A -85,B 0,C 180,E1 -17891.402,E2 -17891.402} C_VEL
LIN {X 0,Y 273.792,Z 737.209,A -85,B 0,C 180,E1 -17893.214,E2 -17893.214} C_VEL
LIN {X 0,Y 272.097,Z 744.892,A -85,B 0,C 180,E1 -17895.413,E2 -17895.413} C_VEL
LIN {X 0,Y 270.586,Z 751.945,A -85,B 0,C 180,E1 -17898.006,E2 -17898.006} C_VEL
LIN {X 0,Y 269.579,Z 756.64,A -85,B 0,C 180,E1 -17900.242,E2 -17900.242} C_VEL
LIN {X 0,Y 268.961,Z 760.225,A -85,B 0,C 180,E1 -17902.492,E2 -17902.492} C_VEL
LIN {X 0,Y 268.669,Z 762.078,A -85,B 0,C 180,E1 -17903.993,E2 -17903.993} C_VEL
LIN {X 0,Y 268.486,Z 763.471,A -85,B 0,C 180,E1 -17905.495,E2 -17905.495} C_VEL
LIN {X 0,Y 268.362,Z 764.463,A -85,B 0,C 180,E1 -17906.996,E2 -17906.996} C_VEL
LIN {X 0,Y 268.21,Z 765.306,A -85,B 0,C 180,E1 -17909.999,E2 -17909.999} C_VEL
LIN {X 0,Y 268.234,Z 765.114,A -85,B 0,C 180,E1 -17911.5,E2 -17911.5} C_VEL
LIN {X 0,Y 268.36,Z 764.529,A -85,B 0,C 180,E1 -17913.001,E2 -17913.001} C_VEL
LIN {X 0,Y 268.482,Z 763.564,A -85,B 0,C 180,E1 -17914.503,E2 -17914.503} C_VEL
LIN {X 0,Y 268.75,Z 761.737,A -85,B 0,C 180,E1 -17916.418,E2 -17916.418} C_VEL
LIN {X 0,Y 269.347,Z 758.145,A -85,B 0,C 180,E1 -17919.006,E2 -17919.006} C_VEL
LIN {X 0,Y 270.182,Z 753.892,A -85,B 0,C 180,E1 -17921.249,E2 -17921.249} C_VEL
LIN {X 0,Y 271.602,Z 747.453,A -85,B 0,C 180,E1 -17923.847,E2 -17923.847} C_VEL
LIN {X 0,Y 273.061,Z 740.375,A -85,B 0,C 180,E1 -17926.061,E2 -17926.061} C_VEL
LIN {X 0,Y 275.102,Z 731.548,A -85,B 0,C 180,E1 -17928.236,E2 -17928.236} C_VEL
LIN {X 0,Y 276.807,Z 722.161,A -85,B 0,C 180,E1 -17930.11,E2 -17930.11} C_VEL
LIN {X 0,Y 278.452,Z 712.466,A -85,B 0,C 180,E1 -17931.66,E2 -17931.66} C_VEL
LIN {X 0,Y 280.269,Z 701.304,A -85,B 0,C 180,E1 -17933.066,E2 -17933.066} C_VEL
LIN {X 0,Y 281.961,Z 688.759,A -85,B 0,C 180,E1 -17934.283,E2 -17934.283} C_VEL
LIN {X 0,Y 283.198,Z 675.811,A -85,B 0,C 180,E1 -17935.197,E2 -17935.197} C_VEL
LIN {X 0,Y 284.161,Z 663.036,A -85,B 0,C 180,E1 -17935.792,E2 -17935.792} C_VEL
LIN {X 0,Y 284.915,Z 640.803,A -85,B 0,C 180,E1 -17936.389,E2 -17936.389} C_VEL
LIN {X 0,Y 286.27,Z 591.107,A -85,B 0,C 180,E1 -17937.626,E2 -17937.626} C_VEL
LIN {X 0,Y 284.966,Z 586.633,A -85,B 0,C 180,E1 -17937.889,E2 -17937.889} C_VEL
LIN {X 0,Y 277.678,Z 568.758,A -85,B 0,C 180,E1 -17939.213,E2 -17939.213} C_VEL
LIN {X 0,Y 271.276,Z 555.197,A -85,B 0,C 180,E1 -17940.432,E2 -17940.432} C_VEL
LIN {X 0,Y 270.289,Z 551.314,A -85,B 0,C 180,E1 -17941.989,E2 -17941.989} C_VEL
LIN {X 0,Y 270.21,Z 550.825,A -85,B 0,C 180,E1 -17942.44,E2 -17942.44} C_VEL
LIN {X 0,Y 270.237,Z 550.816,A -85,B 0,C 180,E1 -17946.736,E2 -17946.736} C_VEL
LIN {X 0,Y 270.171,Z 550.82,A -85,B 0,C 180,E1 -17950.564,E2 -17950.564} C_VEL
LIN {X 0,Y 270.15,Z 550.814,A -85,B 0,C 180,E1 -17954.618,E2 -17954.618} C_VEL
LIN {X 0,Y 270.204,Z 550.821,A -85,B 0,C 180,E1 -17958.961,E2 -17958.961} C_VEL
LIN {X 0,Y 270.209,Z 550.805,A -85,B 0,C 180,E1 -17962.776,E2 -17962.776} C_VEL
LIN {X 0,Y 270.199,Z 550.823,A -85,B 0,C 180,E1 -17966.892,E2 -17966.892} C_VEL
LIN {X 0,Y 270.192,Z 550.826,A -85,B 0,C 180,E1 -17969.225,E2 -17969.225} C_VEL
LIN {X 0,Y 269.523,Z 550.911,A -85,B 0,C 180,E1 -17970.469,E2 -17970.469} C_VEL
LIN {X 0,Y 266.707,Z 551.261,A -85,B 0,C 180,E1 -17972.497,E2 -17972.497} C_VEL
LIN {X 0,Y 264.314,Z 551.561,A -85,B 0,C 180,E1 -17974.145,E2 -17974.145} C_VEL
LIN {X 0,Y 263.274,Z 551.691,A -85,B 0,C 180,E1 -17975.422,E2 -17975.422} C_VEL
LIN {X 0,Y 263.183,Z 551.698,A -85,B 0,C 180,E1 -17975.855,E2 -17975.855} C_VEL
LIN {X 0,Y 263.257,Z 551.689,A -85,B 0,C 180,E1 -17979.693,E2 -17979.693} C_VEL
LIN {X 0,Y 263.344,Z 551.668,A -85,B 0,C 180,E1 -17984.521,E2 -17984.521} C_VEL
LIN {X 0,Y 263.367,Z 551.665,A -85,B 0,C 180,E1 -17989.234,E2 -17989.234} C_VEL
LIN {X 0,Y 263.566,Z 551.652,A -85,B 0,C 180,E1 -17992.338,E2 -17992.338} C_VEL
LIN {X 0,Y 263.745,Z 551.626,A -85,B 0,C 180,E1 -17998.473,E2 -17998.473} C_VEL
LIN {X 0,Y 263.746,Z 551.627,A -85,B 0,C 180,E1 -18001.527,E2 -18001.527} C_VEL
LIN {X 0,Y 263.566,Z 551.652,A -85,B 0,C 180,E1 -18007.662,E2 -18007.662} C_VEL
LIN {X 0,Y 263.367,Z 551.664,A -85,B 0,C 180,E1 -18010.766,E2 -18010.766} C_VEL
LIN {X 0,Y 263.344,Z 551.669,A -85,B 0,C 180,E1 -18015.478,E2 -18015.478} C_VEL
LIN {X 0,Y 263.257,Z 551.688,A -85,B 0,C 180,E1 -18020.307,E2 -18020.307} C_VEL
LIN {X 0,Y 263.201,Z 551.697,A -85,B 0,C 180,E1 -18025.292,E2 -18025.292} C_VEL
LIN {X 0,Y 263.158,Z 551.705,A -85,B 0,C 180,E1 -18028.732,E2 -18028.732} C_VEL
LIN {X 0,Y 263.127,Z 551.708,A -85,B 0,C 180,E1 -18032.289,E2 -18032.289} C_VEL
LIN {X 0,Y 263.177,Z 551.674,A -85,B 0,C 180,E1 -18036.764,E2 -18036.764} C_VEL
LIN {X 0,Y 263.128,Z 551.71,A -85,B 0,C 180,E1 -18039.869,E2 -18039.869} C_VEL
LIN {X 0,Y 263.134,Z 551.7,A -85,B 0,C 180,E1 -18043.982,E2 -18043.982} C_VEL
LIN {X 0,Y 263.206,Z 551.695,A -85,B 0,C 180,E1 -18048.387,E2 -18048.387} C_VEL
LIN {X 0,Y 263.235,Z 551.792,A -85,B 0,C 180,E1 -18052.587,E2 -18052.587} C_VEL
LIN {X 0,Y 265.517,Z 561.596,A -85,B 0,C 180,E1 -18056.646,E2 -18056.646} C_VEL
LIN {X 0,Y 266.968,Z 568.058,A -85,B 0,C 180,E1 -18059.054,E2 -18059.054} C_VEL
LIN {X 0,Y 273.592,Z 583.717,A -85,B 0,C 180,E1 -18060.386,E2 -18060.386} C_VEL
LIN {X 0,Y 275.017,Z 587.946,A -85,B 0,C 180,E1 -18060.678,E2 -18060.678} C_VEL
LIN {X 0,Y 279.185,Z 614.528,A -85,B 0,C 180,E1 -18061.914,E2 -18061.914} C_VEL
LIN {X 0,Y 279.132,Z 623.041,A -85,B 0,C 180,E1 -18062.151,E2 -18062.151} C_VEL
LIN {X 0,Y 277.434,Z 676.544,A -85,B 0,C 180,E1 -18063.534,E2 -18063.534} C_VEL
LIN {X 0,Y 276.333,Z 690.445,A -85,B 0,C 180,E1 -18064.182,E2 -18064.182} C_VEL
LIN {X 0,Y 274.859,Z 702.89,A -85,B 0,C 180,E1 -18065.047,E2 -18065.047} C_VEL
LIN {X 0,Y 273.006,Z 715.587,A -85,B 0,C 180,E1 -18066.284,E2 -18066.284} C_VEL
LIN {X 0,Y 271.042,Z 726.865,A -85,B 0,C 180,E1 -18067.716,E2 -18067.716} C_VEL
LIN {X 0,Y 269.061,Z 737.028,A -85,B 0,C 180,E1 -18069.354,E2 -18069.354} C_VEL
LIN {X 0,Y 267.133,Z 746.534,A -85,B 0,C 180,E1 -18071.285,E2 -18071.285} C_VEL
LIN {X 0,Y 265.3,Z 755.117,A -85,B 0,C 180,E1 -18073.456,E2 -18073.456} C_VEL
LIN {X 0,Y 263.769,Z 762.305,A -85,B 0,C 180,E1 -18075.733,E2 -18075.733} C_VEL
LIN {X 0,Y 262.726,Z 767.156,A -85,B 0,C 180,E1 -18077.644,E2 -18077.644} C_VEL
LIN {X 0,Y 261.908,Z 771.878,A -85,B 0,C 180,E1 -18079.957,E2 -18079.957} C_VEL
LIN {X 0,Y 261.356,Z 775.49,A -85,B 0,C 180,E1 -18082.274,E2 -18082.274} C_VEL
LIN {X 0,Y 261.084,Z 778.348,A -85,B 0,C 180,E1 -18084.866,E2 -18084.866} C_VEL
LIN {X 0,Y 261.063,Z 779.749,A -85,B 0,C 180,E1 -18086.915,E2 -18086.915} C_VEL
LIN {X 0,Y 261.109,Z 780.358,A -85,B 0,C 180,E1 -18088.459,E2 -18088.459} C_VEL
LIN {X 0,Y 261.079,Z 780.682,A -85,B 0,C 180,E1 -18090.58,E2 -18090.58} C_VEL
LIN {X 0,Y 261.105,Z 782.96,A -85,B 0,C 180,E1 -18093.087,E2 -18093.087} C_VEL
LIN {X 0,Y 261.254,Z 783.797,A -85,B 0,C 180,E1 -18095.533,E2 -18095.533} C_VEL
LIN {X 0,Y 261.69,Z 783.291,A -85,B 0,C 180,E1 -18097.718,E2 -18097.718} C_VEL
LIN {X 0,Y 262.21,Z 782.251,A -85,B 0,C 180,E1 -18099.256,E2 -18099.256} C_VEL
LIN {X 0,Y 263.276,Z 779.555,A -85,B 0,C 180,E1 -18101.55,E2 -18101.55} C_VEL
LIN {X 0,Y 264.679,Z 775.539,A -85,B 0,C 180,E1 -18103.827,E2 -18103.827} C_VEL
LIN {X 0,Y 265.727,Z 772.033,A -85,B 0,C 180,E1 -18105.337,E2 -18105.337} C_VEL
LIN {X 0,Y 267.532,Z 766.553,A -85,B 0,C 180,E1 -18107.191,E2 -18107.191} C_VEL
LIN {X 0,Y 269.443,Z 759.75,A -85,B 0,C 180,E1 -18109.03,E2 -18109.03} C_VEL
LIN {X 0,Y 271.29,Z 752.121,A -85,B 0,C 180,E1 -18110.659,E2 -18110.659} C_VEL
LIN {X 0,Y 273.373,Z 742.626,A -85,B 0,C 180,E1 -18112.285,E2 -18112.285} C_VEL
LIN {X 0,Y 275.033,Z 733.345,A -85,B 0,C 180,E1 -18113.534,E2 -18113.534} C_VEL
LIN {X 0,Y 276.553,Z 723.35,A -85,B 0,C 180,E1 -18114.592,E2 -18114.592} C_VEL
LIN {X 0,Y 277.855,Z 710.966,A -85,B 0,C 180,E1 -18115.569,E2 -18115.569} C_VEL
LIN {X 0,Y 279.561,Z 691.125,A -85,B 0,C 180,E1 -18116.704,E2 -18116.704} C_VEL
LIN {X 0,Y 282.952,Z 661.724,A -85,B 0,C 180,E1 -18118.161,E2 -18118.161} C_VEL
LIN {X 0,Y 286.651,Z 632.412,A -85,B 0,C 180,E1 -18119.567,E2 -18119.567} C_VEL
LIN {X 0,Y 290.783,Z 620.133,A -85,B 0,C 180,E1 -18120.77,E2 -18120.77} C_VEL
LIN {X 0,Y 293.303,Z 611.184,A -85,B 0,C 180,E1 -18122.028,E2 -18122.028} C_VEL
LIN {X 0,Y 293.482,Z 609.374,A -85,B 0,C 180,E1 -18122.442,E2 -18122.442} C_VEL
LIN {X 0,Y 293.4,Z 603.869,A -85,B 0,C 180,E1 -18124.177,E2 -18124.177} C_VEL
LIN {X 0,Y 292.715,Z 601.908,A -85,B 0,C 180,E1 -18125.281,E2 -18125.281} C_VEL
LIN {X 0,Y 291.303,Z 599.832,A -85,B 0,C 180,E1 -18127.235,E2 -18127.235} C_VEL
LIN {X 0,Y 290.192,Z 598.617,A -85,B 0,C 180,E1 -18129.196,E2 -18129.196} C_VEL
LIN {X 0,Y 289.434,Z 598.03,A -85,B 0,C 180,E1 -18131.172,E2 -18131.172} C_VEL
LIN {X 0,Y 289.029,Z 598.14,A -85,B 0,C 180,E1 -18133.157,E2 -18133.157} C_VEL
LIN {X 0,Y 288.898,Z 598.873,A -85,B 0,C 180,E1 -18135.131,E2 -18135.131} C_VEL
LIN {X 0,Y 288.959,Z 601.365,A -85,B 0,C 180,E1 -18138.002,E2 -18138.002} C_VEL
LIN {X 0,Y 289.203,Z 603.914,A -85,B 0,C 180,E1 -18139.983,E2 -18139.983} C_VEL
LIN {X 0,Y 289.515,Z 608.593,A -85,B 0,C 180,E1 -18142.636,E2 -18142.636} C_VEL
LIN {X 0,Y 289.556,Z 613.555,A -85,B 0,C 180,E1 -18144.803,E2 -18144.803} C_VEL
LIN {X 0,Y 289.386,Z 614.757,A -85,B 0,C 180,E1 -18145.209,E2 -18145.209} C_VEL
LIN {X 0,Y 283.995,Z 632.739,A -85,B 0,C 180,E1 -18149.602,E2 -18149.602} C_VEL
LIN {X 0,Y 285.991,Z 646.766,A -85,B 0,C 180,E1 -18151.415,E2 -18151.415} C_VEL
LIN {X 0,Y 287.49,Z 659.723,A -85,B 0,C 180,E1 -18152.82,E2 -18152.82} C_VEL
LIN {X 0,Y 287.944,Z 667.529,A -85,B 0,C 180,E1 -18153.501,E2 -18153.501} C_VEL
LIN {X 0,Y 283.259,Z 708.736,A -85,B 0,C 180,E1 -18155.395,E2 -18155.395} C_VEL
LIN {X 0,Y 281.647,Z 719.084,A -85,B 0,C 180,E1 -18156.078,E2 -18156.078} C_VEL
LIN {X 0,Y 279.572,Z 729.667,A -85,B 0,C 180,E1 -18157.068,E2 -18157.068} C_VEL
LIN {X 0,Y 277.263,Z 739.35,A -85,B 0,C 180,E1 -18158.24,E2 -18158.24} C_VEL
LIN {X 0,Y 274.519,Z 749.044,A -85,B 0,C 180,E1 -18159.781,E2 -18159.781} C_VEL
LIN {X 0,Y 272.396,Z 756,A -85,B 0,C 180,E1 -18161.185,E2 -18161.185} C_VEL
LIN {X 0,Y 269.959,Z 763.065,A -85,B 0,C 180,E1 -18162.97,E2 -18162.97} C_VEL
LIN {X 0,Y 267.75,Z 768.533,A -85,B 0,C 180,E1 -18164.783,E2 -18164.783} C_VEL
LIN {X 0,Y 265.613,Z 773.595,A -85,B 0,C 180,E1 -18167.003,E2 -18167.003} C_VEL
LIN {X 0,Y 263.955,Z 777.144,A -85,B 0,C 180,E1 -18169.258,E2 -18169.258} C_VEL
LIN {X 0,Y 263.046,Z 778.738,A -85,B 0,C 180,E1 -18170.775,E2 -18170.775} C_VEL
LIN {X 0,Y 262.404,Z 779.721,A -85,B 0,C 180,E1 -18172.304,E2 -18172.304} C_VEL
LIN {X 0,Y 261.854,Z 780.134,A -85,B 0,C 180,E1 -18173.837,E2 -18173.837} C_VEL
LIN {X 0,Y 261.408,Z 779.99,A -85,B 0,C 180,E1 -18175.374,E2 -18175.374} C_VEL
LIN {X 0,Y 261.199,Z 779.288,A -85,B 0,C 180,E1 -18176.915,E2 -18176.915} C_VEL
LIN {X 0,Y 261.114,Z 778.018,A -85,B 0,C 180,E1 -18178.458,E2 -18178.458} C_VEL
LIN {X 0,Y 261.068,Z 774.958,A -85,B 0,C 180,E1 -18180.771,E2 -18180.771} C_VEL
LIN {X 0,Y 261.269,Z 770.423,A -85,B 0,C 180,E1 -18183.084,E2 -18183.084} C_VEL
LIN {X 0,Y 261.408,Z 765.264,A -85,B 0,C 180,E1 -18184.983,E2 -18184.983} C_VEL
LIN {X 0,Y 261.726,Z 758.529,A -85,B 0,C 180,E1 -18186.94,E2 -18186.94} C_VEL
LIN {X 0,Y 262.186,Z 749.92,A -85,B 0,C 180,E1 -18188.867,E2 -18188.867} C_VEL
LIN {X 0,Y 262.556,Z 742.37,A -85,B 0,C 180,E1 -18190.215,E2 -18190.215} C_VEL
LIN {X 0,Y 263.057,Z 733.089,A -85,B 0,C 180,E1 -18191.559,E2 -18191.559} C_VEL
LIN {X 0,Y 263.605,Z 722.586,A -85,B 0,C 180,E1 -18192.706,E2 -18192.706} C_VEL
LIN {X 0,Y 263.995,Z 712.211,A -85,B 0,C 180,E1 -18193.568,E2 -18193.568} C_VEL
LIN {X 0,Y 264.395,Z 700.208,A -85,B 0,C 180,E1 -18194.234,E2 -18194.234} C_VEL
LIN {X 0,Y 265.372,Z 654.449,A -85,B 0,C 180,E1 -18196.18,E2 -18196.18} C_VEL
LIN {X 0,Y 263.971,Z 632.743,A -85,B 0,C 180,E1 -18197.129,E2 -18197.129} C_VEL
LIN {X 0,Y 264.002,Z 631.799,A -85,B 0,C 180,E1 -18197.227,E2 -18197.227} C_VEL
LIN {X 0,Y 265.434,Z 612.55,A -85,B 0,C 180,E1 -18201.35,E2 -18201.35} C_VEL
LIN {X 0,Y 266.961,Z 593.975,A -85,B 0,C 180,E1 -18205.328,E2 -18205.328} C_VEL
LIN {X 0,Y 268.419,Z 576.978,A -85,B 0,C 180,E1 -18208.972,E2 -18208.972} C_VEL
LIN {X 0,Y 265.631,Z 563.15,A -85,B 0,C 180,E1 -18212.149,E2 -18212.149} C_VEL
LIN {X 0,Y 263.242,Z 551.885,A -85,B 0,C 180,E1 -18214.871,E2 -18214.871} C_VEL
LIN {X 0,Y 263.165,Z 551.705,A -85,B 0,C 180,E1 -18217.896,E2 -18217.896} C_VEL
LIN {X 0,Y 263.129,Z 551.659,A -85,B 0,C 180,E1 -18221.893,E2 -18221.893} C_VEL
LIN {X 0,Y 263.14,Z 551.703,A -85,B 0,C 180,E1 -18226.148,E2 -18226.148} C_VEL
LIN {X 0,Y 263.116,Z 551.674,A -85,B 0,C 180,E1 -18230.128,E2 -18230.128} C_VEL
LIN {X 0,Y 263.167,Z 551.701,A -85,B 0,C 180,E1 -18234.017,E2 -18234.017} C_VEL
LIN {X 0,Y 263.184,Z 551.852,A -85,B 0,C 180,E1 -18237.264,E2 -18237.264} C_VEL
LIN {X 0,Y 264.029,Z 555.236,A -85,B 0,C 180,E1 -18238.737,E2 -18238.737} C_VEL
LIN {X 0,Y 266.264,Z 560.024,A -85,B 0,C 180,E1 -18239.255,E2 -18239.255} C_VEL
LIN {X 0,Y 273.682,Z 575.885,A -85,B 0,C 180,E1 -18240.653,E2 -18240.653} C_VEL
LIN {X 0,Y 279.848,Z 591.756,A -85,B 0,C 180,E1 -18241.821,E2 -18241.821} C_VEL
LIN {X 0,Y 278.565,Z 639.446,A -85,B 0,C 180,E1 -18243.041,E2 -18243.041} C_VEL
LIN {X 0,Y 277.702,Z 662.671,A -85,B 0,C 180,E1 -18243.66,E2 -18243.66} C_VEL
LIN {X 0,Y 276.674,Z 676.403,A -85,B 0,C 180,E1 -18244.314,E2 -18244.314} C_VEL
LIN {X 0,Y 275.449,Z 688.714,A -85,B 0,C 180,E1 -18245.202,E2 -18245.202} C_VEL
LIN {X 0,Y 273.86,Z 700.514,A -85,B 0,C 180,E1 -18246.359,E2 -18246.359} C_VEL
LIN {X 0,Y 271.966,Z 711.859,A -85,B 0,C 180,E1 -18247.793,E2 -18247.793} C_VEL
LIN {X 0,Y 270.239,Z 721.431,A -85,B 0,C 180,E1 -18249.322,E2 -18249.322} C_VEL
LIN {X 0,Y 268.396,Z 731.241,A -85,B 0,C 180,E1 -18251.289,E2 -18251.289} C_VEL
LIN {X 0,Y 266.341,Z 740.151,A -85,B 0,C 180,E1 -18253.52,E2 -18253.52} C_VEL
LIN {X 0,Y 264.786,Z 747.316,A -85,B 0,C 180,E1 -18255.786,E2 -18255.786} C_VEL
LIN {X 0,Y 263.647,Z 752.151,A -85,B 0,C 180,E1 -18257.686,E2 -18257.686} C_VEL
LIN {X 0,Y 262.589,Z 756.846,A -85,B 0,C 180,E1 -18259.98,E2 -18259.98} C_VEL
LIN {X 0,Y 261.925,Z 760.431,A -85,B 0,C 180,E1 -18262.289,E2 -18262.289} C_VEL
LIN {X 0,Y 261.602,Z 762.283,A -85,B 0,C 180,E1 -18263.83,E2 -18263.83} C_VEL
LIN {X 0,Y 261.4,Z 763.677,A -85,B 0,C 180,E1 -18265.372,E2 -18265.372} C_VEL
LIN {X 0,Y 261.277,Z 764.668,A -85,B 0,C 180,E1 -18266.915,E2 -18266.915} C_VEL
LIN {X 0,Y 261.136,Z 765.51,A -85,B 0,C 180,E1 -18269.999,E2 -18269.999} C_VEL
LIN {X 0,Y 261.164,Z 765.318,A -85,B 0,C 180,E1 -18271.541,E2 -18271.541} C_VEL
LIN {X 0,Y 261.275,Z 764.733,A -85,B 0,C 180,E1 -18273.082,E2 -18273.082} C_VEL
LIN {X 0,Y 261.6,Z 762.413,A -85,B 0,C 180,E1 -18276.168,E2 -18276.168} C_VEL
LIN {X 0,Y 262.114,Z 759.545,A -85,B 0,C 180,E1 -18278.479,E2 -18278.479} C_VEL
LIN {X 0,Y 262.873,Z 755.654,A -85,B 0,C 180,E1 -18280.785,E2 -18280.785} C_VEL
LIN {X 0,Y 264.014,Z 750.637,A -85,B 0,C 180,E1 -18283.076,E2 -18283.076} C_VEL
LIN {X 0,Y 265.38,Z 744.319,A -85,B 0,C 180,E1 -18285.355,E2 -18285.355} C_VEL
LIN {X 0,Y 267.238,Z 736.403,A -85,B 0,C 180,E1 -18287.602,E2 -18287.602} C_VEL
LIN {X 0,Y 269.047,Z 728.334,A -85,B 0,C 180,E1 -18289.453,E2 -18289.453} C_VEL
LIN {X 0,Y 270.824,Z 718.492,A -85,B 0,C 180,E1 -18291.302,E2 -18291.302} C_VEL
LIN {X 0,Y 272.766,Z 707.41,A -85,B 0,C 180,E1 -18292.935,E2 -18292.935} C_VEL
LIN {X 0,Y 274.499,Z 696.536,A -85,B 0,C 180,E1 -18294.181,E2 -18294.181} C_VEL
LIN {X 0,Y 276.002,Z 684.512,A -85,B 0,C 180,E1 -18295.245,E2 -18295.245} C_VEL
LIN {X 0,Y 277.139,Z 672.157,A -85,B 0,C 180,E1 -18296.04,E2 -18296.04} C_VEL
LIN {X 0,Y 278.004,Z 659.337,A -85,B 0,C 180,E1 -18296.559,E2 -18296.559} C_VEL
LIN {X 0,Y 279.968,Z 592.259,A -85,B 0,C 180,E1 -18298.275,E2 -18298.275} C_VEL
LIN {X 0,Y 275.546,Z 580.419,A -85,B 0,C 180,E1 -18299.121,E2 -18299.121} C_VEL
LIN {X 0,Y 268.941,Z 565.518,A -85,B 0,C 180,E1 -18300.365,E2 -18300.365} C_VEL
LIN {X 0,Y 264.092,Z 555.533,A -85,B 0,C 180,E1 -18301.342,E2 -18301.342} C_VEL
LIN {X 0,Y 263.496,Z 553.166,A -85,B 0,C 180,E1 -18302.237,E2 -18302.237} C_VEL
LIN {X 0,Y 263.17,Z 551.724,A -85,B 0,C 180,E1 -18303.019,E2 -18303.019} C_VEL
LIN {X 0,Y 263.201,Z 551.693,A -85,B 0,C 180,E1 -18306.768,E2 -18306.768} C_VEL
LIN {X 0,Y 263.111,Z 551.696,A -85,B 0,C 180,E1 -18309.869,E2 -18309.869} C_VEL
LIN {X 0,Y 263.119,Z 551.693,A -85,B 0,C 180,E1 -18313.983,E2 -18313.983} C_VEL
LIN {X 0,Y 263.143,Z 551.706,A -85,B 0,C 180,E1 -18318.399,E2 -18318.399} C_VEL
LIN {X 0,Y 263.183,Z 551.673,A -85,B 0,C 180,E1 -18322.107,E2 -18322.107} C_VEL
LIN {X 0,Y 263.178,Z 551.702,A -85,B 0,C 180,E1 -18325.889,E2 -18325.889} C_VEL
LIN {X 0,Y 263.145,Z 551.707,A -85,B 0,C 180,E1 -18329.506,E2 -18329.506} C_VEL
LIN {X 0,Y 263.187,Z 551.69,A -85,B 0,C 180,E1 -18333.002,E2 -18333.002} C_VEL
LIN {X 0,Y 263.183,Z 551.698,A -85,B 0,C 180,E1 -18335.855,E2 -18335.855} C_VEL
LIN {X 0,Y 262.498,Z 551.781,A -85,B 0,C 180,E1 -18337.132,E2 -18337.132} C_VEL
LIN {X 0,Y 259.658,Z 552.14,A -85,B 0,C 180,E1 -18339.214,E2 -18339.214} C_VEL
LIN {X 0,Y 257.276,Z 552.438,A -85,B 0,C 180,E1 -18340.907,E2 -18340.907} C_VEL
LIN {X 0,Y 256.278,Z 552.555,A -85,B 0,C 180,E1 -18342.219,E2 -18342.219} C_VEL
LIN {X 0,Y 256.208,Z 552.56,A -85,B 0,C 180,E1 -18342.664,E2 -18342.664} C_VEL
LIN {X 0,Y 256.249,Z 552.56,A -85,B 0,C 180,E1 -18345.709,E2 -18345.709} C_VEL
LIN {X 0,Y 256.473,Z 552.52,A -85,B 0,C 180,E1 -18350.56,E2 -18350.56} C_VEL
LIN {X 0,Y 256.481,Z 552.537,A -85,B 0,C 180,E1 -18353.707,E2 -18353.707} C_VEL
LIN {X 0,Y 256.708,Z 552.501,A -85,B 0,C 180,E1 -18358.431,E2 -18358.431} C_VEL
LIN {X 0,Y 256.708,Z 552.503,A -85,B 0,C 180,E1 -18361.569,E2 -18361.569} C_VEL
LIN {X 0,Y 256.533,Z 552.526,A -85,B 0,C 180,E1 -18367.873,E2 -18367.873} C_VEL
LIN {X 0,Y 256.303,Z 552.545,A -85,B 0,C 180,E1 -18371.066,E2 -18371.066} C_VEL
LIN {X 0,Y 256.293,Z 552.545,A -85,B 0,C 180,E1 -18375.915,E2 -18375.915} C_VEL
LIN {X 0,Y 256.161,Z 552.568,A -85,B 0,C 180,E1 -18380.896,E2 -18380.896} C_VEL
LIN {X 0,Y 256.181,Z 552.573,A -85,B 0,C 180,E1 -18385.139,E2 -18385.139} C_VEL
LIN {X 0,Y 256.097,Z 552.584,A -85,B 0,C 180,E1 -18389.602,E2 -18389.602} C_VEL
LIN {X 0,Y 256.062,Z 552.59,A -85,B 0,C 180,E1 -18393.294,E2 -18393.294} C_VEL
LIN {X 0,Y 256.109,Z 552.557,A -85,B 0,C 180,E1 -18397.272,E2 -18397.272} C_VEL
LIN {X 0,Y 256.076,Z 552.575,A -85,B 0,C 180,E1 -18401.199,E2 -18401.199} C_VEL
LIN {X 0,Y 256.071,Z 552.585,A -85,B 0,C 180,E1 -18405.527,E2 -18405.527} C_VEL
LIN {X 0,Y 256.127,Z 552.582,A -85,B 0,C 180,E1 -18408.813,E2 -18408.813} C_VEL
LIN {X 0,Y 256.184,Z 552.737,A -85,B 0,C 180,E1 -18411.859,E2 -18411.859} C_VEL
LIN {X 0,Y 258.574,Z 562.726,A -85,B 0,C 180,E1 -18416.141,E2 -18416.141} C_VEL
LIN {X 0,Y 259.668,Z 567.649,A -85,B 0,C 180,E1 -18418.054,E2 -18418.054} C_VEL
LIN {X 0,Y 262.147,Z 573.433,A -85,B 0,C 180,E1 -18418.643,E2 -18418.643} C_VEL
LIN {X 0,Y 268.649,Z 588.718,A -85,B 0,C 180,E1 -18419.941,E2 -18419.941} C_VEL
LIN {X 0,Y 271.742,Z 607.184,A -85,B 0,C 180,E1 -18420.863,E2 -18420.863} C_VEL
LIN {X 0,Y 273.067,Z 617.672,A -85,B 0,C 180,E1 -18421.324,E2 -18421.324} C_VEL
LIN {X 0,Y 271.107,Z 676.354,A -85,B 0,C 180,E1 -18422.867,E2 -18422.867} C_VEL
LIN {X 0,Y 269.966,Z 690.25,A -85,B 0,C 180,E1 -18423.526,E2 -18423.526} C_VEL
LIN {X 0,Y 268.579,Z 701.58,A -85,B 0,C 180,E1 -18424.318,E2 -18424.318} C_VEL
LIN {X 0,Y 266.781,Z 713.802,A -85,B 0,C 180,E1 -18425.488,E2 -18425.488} C_VEL
LIN {X 0,Y 264.712,Z 725.37,A -85,B 0,C 180,E1 -18426.947,E2 -18426.947} C_VEL
LIN {X 0,Y 262.598,Z 735.787,A -85,B 0,C 180,E1 -18428.616,E2 -18428.616} C_VEL
LIN {X 0,Y 260.747,Z 744.664,A -85,B 0,C 180,E1 -18430.395,E2 -18430.395} C_VEL
LIN {X 0,Y 258.813,Z 753.554,A -85,B 0,C 180,E1 -18432.622,E2 -18432.622} C_VEL
LIN {X 0,Y 257.095,Z 760.985,A -85,B 0,C 180,E1 -18434.95,E2 -18434.95} C_VEL
LIN {X 0,Y 255.752,Z 766.952,A -85,B 0,C 180,E1 -18437.302,E2 -18437.302} C_VEL
LIN {X 0,Y 254.876,Z 771.673,A -85,B 0,C 180,E1 -18439.676,E2 -18439.676} C_VEL
LIN {X 0,Y 254.315,Z 775.286,A -85,B 0,C 180,E1 -18442.059,E2 -18442.059} C_VEL
LIN {X 0,Y 253.99,Z 778.347,A -85,B 0,C 180,E1 -18444.963,E2 -18444.963} C_VEL
LIN {X 0,Y 253.962,Z 779.544,A -85,B 0,C 180,E1 -18446.829,E2 -18446.829} C_VEL
LIN {X 0,Y 254.015,Z 780.153,A -85,B 0,C 180,E1 -18448.416,E2 -18448.416} C_VEL
LIN {X 0,Y 254.009,Z 780.32,A -85,B 0,C 180,E1 -18450.794,E2 -18450.794} C_VEL
LIN {X 0,Y 254.025,Z 782.585,A -85,B 0,C 180,E1 -18453.173,E2 -18453.173} C_VEL
LIN {X 0,Y 254.168,Z 783.591,A -85,B 0,C 180,E1 -18455.475,E2 -18455.475} C_VEL
LIN {X 0,Y 254.314,Z 783.735,A -85,B 0,C 180,E1 -18456.348,E2 -18456.348} C_VEL
